// TwinCAT 3 PLC project External_Conveyor_system
// ProgramVersion: 3.1.4026.19
// libraries:
//   Tc2_EtherCAT, * (Beckhoff Automation GmbH)
//   Tc2_MC2, * (Beckhoff Automation GmbH)
//   Tc2_Standard, * (Beckhoff Automation GmbH)
//   Tc2_System, * (Beckhoff Automation GmbH)
//   Tc2_Utilities, * (Beckhoff Automation GmbH)
//   Tc3_Database, * (Beckhoff Automation GmbH)
//   Tc3_EventLogger, * (Beckhoff Automation GmbH)
//   Tc3_JsonXml, * (Beckhoff Automation GmbH)
//   Tc3_Module, * (Beckhoff Automation GmbH)
// project tree:
//   DUTs/EtherCAT模組/ MM540_Raw.TcDUT
//   DUTs/JOG用元素/ e_Site_Select.TcTLEO
//   DUTs/工單結構/ WorkOrder_Data.TcDUT
//   DUTs/變頻器IO/ VFD_E_IO.TcDUT
//   GVLs/ Axis.TcGVL, Config.TcGVL, Hmi_Web.TcGVL, Input.TcGVL, IO.TcGVL, Output.TcGVL, ProjectData.TcGVL, Safety.TcGVL
//   MSG/訊息列表/ MsgBuff.TcGVL
//   MSG/訊息格式/ MsgLevel.TcDUT, MsgStruct.TcDUT, MsgStruct_RAW.TcDUT
//   MSG/通知訊息/ MsgMain.TcPOU, MsgPush.TcPOU, uuidv7_g.TcPOU
//   / Note.TcPOU (excluded from build), PlcTask.TcTTO
//   POUs/ MAIN.TcPOU
//   POUs/功能塊/ ErrorCodeConver.TcPOU, pMsg.TcPOU, RW_Config.TcPOU
//   POUs/功能塊/EtherCat相關/ EtherCat_Driver_Reset.TcPOU, GetEtherSta.TcPOU
//   POUs/功能塊/字串處理功能塊/字串填充/ FILLSTRING.TcPOU
//   POUs/功能塊/字串處理功能塊/字串記憶/ WStrMem.TcPOU
//   POUs/功能塊/字串處理功能塊/字串連接/ StrConcat.TcPOU, WStrConcat.TcPOU
//   POUs/功能塊/資料庫 Postgre相關/動作資料/ ReadSQLData.TcPOU
//   POUs/功能塊/資料庫 Postgre相關/動作資料/相關結構/ e_db_steel_local.TcTLEO, e_db_steel_status.TcTLEO (not stored), sc_db_Set_Work_Order_WaitLoading_Pos.TcDUT, sc_db_Steel_Status.TcDUT
//   POUs/功能塊/資料庫 Postgre相關/記錄用/程式紀錄/ StepLog_Struct.TcDUT, Step_Log.TcPOU
//   POUs/動作流程控制/ Alignment_pos.TcDUT, FeedMain.TcPOU
//   POUs/動作流程控制/滾輪整料/ PullOver.TcPOU
//   POUs/安全控制/ MaBaseState.TcPOU
//   POUs/硬體控制/ AxisAction.TcPOU
//   POUs/硬體控制/出料滾輪/ ProductRoller.TcPOU
//   POUs/硬體控制/測高/ AxisBase.TcPOU, HeightMeasurer.TcPOU
//   POUs/硬體控制/油壓系統/ Hydraulic.TcPOU, Hydraulic_Action.TcDUT
//   POUs/硬體控制/測寬/ I_DisSensor.TcIO, OGD251_Decoder.TcPOU, Sensor.TcPOU
//   POUs/硬體控制/台車/ ActionMode.TcDUT, Axis_VFD.TcPOU, I_Axis.TcIO
//   POUs/硬體控制/台車/編碼器/ MM540.TcPOU
//   POUs/硬體控制/定位柱/ StopPin.TcPOU
//   POUs/硬體控制/進料滾輪/ FeedRoller.TcPOU
//   POUs/資料轉換/ HMI_WEB_dataConver.TcPOU
// (motion and I/O tree: see PLC project main)
// real-time tasks:
//   TASK Main_IO_Task: cycle T#2ms, priority 6, ADS port 353
//   TASK PlcTask: cycle T#10ms, priority 14, ADS port 350
//   TASK Conveyor: cycle T#10ms, priority 22, ADS port 355
// variable links:

CONFIGURATION External_Conveyor_system
    RESOURCE PLC ON TwinCAT3
        TASK PlcTask(INTERVAL := T#10ms, PRIORITY := 22);
        PROGRAM MAIN WITH PlcTask : MAIN;
    END_RESOURCE
END_CONFIGURATION

// ---- DUTs/EtherCAT模組/MM540_Raw.TcDUT
TYPE MM540_Raw :
STRUCT
	// 編碼器位置
	Inc AT %I*					: DINT;
	
	// 編碼器重設狀態
	Inc_Preload_Done AT %I*		: BOOL;
	
	// 編碼器 A相 錯誤
	Inc_Error_A AT %I*			: BOOL;
	
	// 編碼器 B相 錯誤
	Inc_Error_B AT %I*			: BOOL;
	
	// 編碼器 C相 錯誤
	Inc_Error_C AT %I*			: BOOL;
	
	// 編碼器1 AB相 錯誤
	Inc_Error_AB AT %I*			: BOOL;
	
	
	// 編碼器設定數值
	Inc_Preload_Value AT %Q*			: DINT;
	(*
	設定數值方式:
	0: Disabled
	1: Preload now
	2: Preload with next 0- impulse
	3: Preload with next DI0 rising edge
	4: Preload with next DI1 rising edge
	5: Preload with next DI2 rising edge
	6: Preload with next DI3 rising edge
	7: Preload with next DI0 falling edge
	8: Preload with next DI1 falling edge
	9: Preload with next DI2 falling edge
	10: Preload with next DI3 falling edge
	>10: Disabled
	*)
	// 編碼器1 設定數值方式
	Inc_Preload_Trigger AT %Q*				: USINT;
	
	// 1:數據無效 0:數據有效
	WcState AT %I*					: BOOL;
	
	// EtherCAT 狀態
	State AT %I*:UINT;
	
	// AMS位置
	addr 	AT %I*					: AMSADDR;
END_STRUCT
END_TYPE

// ---- DUTs/JOG用元素/e_Site_Select.TcTLEO
{attribute 'qualified_only'}
{attribute 'strict'}
{attribute 'to_string'}
TYPE e_Jog_Site_Select :
(
	Input_site := 0,
	Output_Site := 1
) INT ;
END_TYPE

// ---- DUTs/工單結構/WorkOrder_Data.TcDUT
// 專案資料結構
TYPE WorkOrder_Data :
STRUCT
	// 加工順序
	SN			: DINT;
	// 高
	Height		: LREAL;
	// 寬
	Width		: LREAL;
	// 素材編號 (uuid)
	steel_id	: STRING(36);
	//  在料架上等待的位置
	waitLoading_pos : LREAL;
END_STRUCT
END_TYPE

// ---- DUTs/變頻器IO/VFD_E_IO.TcDUT
TYPE VFD_E_IO :
STRUCT
	// 正轉 Output
	o_FWD : POINTER TO BOOL;
	
	// 逆轉 Output
	o_REV : POINTER TO BOOL;
	
	// 速度bit1 Output
	o_Speed1 : POINTER TO BOOL;
	
	// 速度bit2 Output
	o_Speed2 : POINTER TO BOOL;
	
	// 速度bit3 Output
	o_Speed3 : POINTER TO BOOL;
	
	// 重置 Output
	o_Reset : POINTER TO BOOL;
	
	// 運行中 Input
	i_Run : POINTER TO BOOL;
	
	// 發生錯誤 Input
	i_Error : POINTER TO BOOL;
END_STRUCT
END_TYPE

// ---- MSG/訊息格式/MsgLevel.TcDUT
{attribute 'qualified_only'}
{attribute 'strict'}
TYPE MsgLevel :
(
	Error	:= 4,
	Alarm	:= 2,
	Info	:= 1,
	None	:= 0
	
)INT;
END_TYPE

// ---- MSG/訊息格式/MsgStruct.TcDUT
{attribute 'pack_mode' := '1'} 
TYPE MsgStruct :
STRUCT
	// 訊息時間
	msgTIME		: DATE_AND_TIME;
	// 訊息等級
	Level		: MsgLevel;
	// 訊息號碼
	Number	: UINT;
	// 訊息附帶文字1
	MsgStr1	: WSTRING(80);
	// 訊息附帶文字2
	MsgStr2	: WSTRING(80);
	// 訊息全文
	raw_msg_str	: WSTRING(250);
END_STRUCT
END_TYPE

// ---- MSG/訊息格式/MsgStruct_RAW.TcDUT
{attribute 'pack_mode' := '1'} 
TYPE MsgStruct_RAW :
STRUCT
	// 訊息時間
	msgTIME		: DATE_AND_TIME;
	// 訊息等級
	Level		: MsgLevel;
	// 訊息號碼
	Number	: UINT;
	// 訊息附帶文字1
	MsgStr1	:  ARRAY[0..159] OF BYTE;
	// 訊息附帶文字2
	MsgStr2	: ARRAY[0..159] OF BYTE;
	// 訊息全文
	raw_msg_str	: ARRAY[0..499] OF BYTE;
END_STRUCT
END_TYPE

// ---- POUs/功能塊/資料庫 Postgre相關/動作資料/相關結構/e_db_steel_local.TcTLEO
{attribute 'qualified_only'}
{attribute 'strict'}
{attribute 'to_string'}
TYPE e_db_steel_local :
(
	holdingEntranceRack := 1, // 吊掛入料區
	entranceRack := 2, // 入料區
	machine := 10, // 機台內
	holdingExitRack := 20, // 吊掛出料區
	exitRack := 21 // 出料區
);
END_TYPE
//  exitRack = '21 '

// ---- POUs/功能塊/資料庫 Postgre相關/動作資料/相關結構/sc_db_Set_Work_Order_WaitLoading_Pos.TcDUT
TYPE sc_db_Set_Work_Order_WaitLoading_Pos :
STRUCT
	uuid : STRING(36);
	Pos : LREAL;
END_STRUCT
END_TYPE

// ---- POUs/功能塊/資料庫 Postgre相關/動作資料/相關結構/sc_db_Steel_Status.TcDUT
TYPE sc_db_Steel_Status :
STRUCT
	uuid : STRING(36);
	steel_status : STRING(80);
	steel_location : STRING(80);
END_STRUCT
END_TYPE

// ---- POUs/功能塊/資料庫 Postgre相關/記錄用/程式紀錄/StepLog_Struct.TcDUT
TYPE StepLog_Struct :
STRUCT
	step_number : DINT;
	created_at : LINT;
	program_name : STRING(80);
	extras_Srt : STRING(255) := '{}';
END_STRUCT
END_TYPE

// ---- POUs/動作流程控制/Alignment_pos.TcDUT
// 排列位置
TYPE Alignment_pos :
STRUCT
	// 分料開始位置 (搬運完成但未分料位置)
	Start : LREAL;
	// 分料結束位置 (推至分料位置)
	End : LREAL;
END_STRUCT
END_TYPE

// ---- POUs/硬體控制/油壓系統/Hydraulic_Action.TcDUT
{attribute 'qualified_only'}
{attribute 'strict'}
TYPE Hydraulic_Action :
(
	DoNothing	:= 0,
	Car_2_Up	:= 1,
	Car_2_Mid	:= 2,
	Car_2_Dn	:= 3,
	Pull_over	:= 4,
	UnPull		:= 5,
	Pull_over_Jog	:= 10
);
END_TYPE

// ---- POUs/硬體控制/台車/ActionMode.TcDUT
{attribute 'qualified_only'}
{attribute 'strict'}
TYPE ActionMode :
(
	DoNothing	:= 0,
	AbsMove		:= 1,
	RelMove		:= 2,
	Home		:= 3,
	Find		:= 4
);
END_TYPE

// ---- GVLs/Axis.TcGVL
VAR_GLOBAL
	
// 軸控制
// ============== 滾輪軸 ==============
	//  進料台車IO
	FeedCar_INV : VFD_E_IO;
	//  進料編碼器
	FeedCar_Enc : MM540;
	
	FeedCar : Axis_VFD;

// ============== 測高軸 ==============
	Axis_StepMoter: AXIS_REF;
	
	Axis_H_Measure: AxisBase;
	
	Override: LREAL := 100;
END_VAR

// ---- GVLs/Config.TcGVL
{attribute 'qualified_only'}
VAR_GLOBAL PERSISTENT
	// 靠邊感應器位置 
	SensorPos : ARRAY [0..15] OF UDINT := [2300,999999,6080,10230];

(* ===============台車===============*)
	// 台車間距
	Car_SetupPos : ARRAY [0..15] OF UDINT := [0,3700,7450,11200];
	
	// 臺車搬移平台寬度 1095mm
	FeedCar_Length : LREAL := 1095;
	
	// 臺車勾板寬度 25mm
	FeedCar_Pin_Length : LREAL := 25;
	
	// 台車橫移的編碼器比例
	FeedCar_Enc_Scal 			: LREAL := -0.025;
	
	// 臺車編碼器原點偏移 (編碼器值)
	FeedCar_Enc_Origin_offset 	: DINT := -880;
	
	// 臺車移動 高速 -> 中速 距離
	dis_to_MidSpeed : LREAL := 470;
	
	// 臺車移動 高速 -> 中速 距離
	dis_to_LowSpeed : LREAL := 80;
	
	// 臺車勾點-整料圓柱 位置  (測量寬度用)
	pos_CarPin_StopPoint		: LREAL := 1120;
	
	// 台車起點 (進料位置)
	pos_StartPoint				: LREAL := 60;
	
	// 台車 等待投料位置 (排列起點)
	pos_Workpiace_StanbyPoint	: LREAL := 1400;
	
	// 台車 投料位置 
	pos_Workpiace_FeedPoint	: LREAL := 2700;
	
	// 材料排列 間距
	dis_Alignment 				: LREAL := 100;
	
	// 材料容許誤差 倍率 (0-1 = 0 ~ 100%) 預設 10%
	Workpiace_Err_size 				: LREAL := 0.1;
	
(* =============== 測高 =============== *)
	// 高基準面位置
	H_Measure_ZeroPoint : LREAL := 642.62;
	
(* =============== 測寬感應器 =============== *)
	// 寬基準面位置
	W_Measure_ZeroPoint : LREAL := 1253;
	
	

END_VAR

// ---- GVLs/Hmi_Web.TcGVL
{attribute 'qualified_only'}
VAR_GLOBAL
(*==================== Jog模式====================*)
	// 料架選擇
	Site_Select : e_Jog_Site_Select;
	
	// 料架速度 (0:高速 1:低速)
	Speed_Select : INT;
	
	// 指定橫移料架
	Module_Select : INT;
	
	// 動力滾輪正轉反饋
	Roller_Fwd_S : BOOL;
	// 動力滾輪反轉反饋
	Roller_Rev_S : BOOL;
	
	// 動力滾輪正轉
	Roller_Fwd : BOOL;
	// 動力滾輪反轉
	Roller_Rev : BOOL;
	
	
	// 動力滾輪上升
	Roller_Up_S : BOOL;
	// 動力滾輪下降
	Roller_Down_S : BOOL;
	
	// 動力滾輪上升
	Roller_Up : BOOL;
	// 動力滾輪下降
	Roller_Down : BOOL;
	
	// 橫移台車位置
	Car_Pos : LREAL;
	// 橫移台車正轉
	Car_Fwd_S : BOOL;
	// 橫移台車反轉
	Car_Rev_S : BOOL;
	
	// 橫移台車正轉
	Car_Fwd : BOOL;
	// 橫移台車反轉
	Car_Rev : BOOL;
	
	
	// 橫移台車上升
	Car_Up_S : BOOL;
	// 橫移台車下降
	Car_Down_S : BOOL;
	
	// 橫移台車上升
	Car_Up : BOOL;
	// 橫移台車下降
	Car_Down : BOOL;
	
	
	// 定位柱上升
	StopPin_Up_S : BOOL;
	// 定位柱下降
	StopPin_Down_S : BOOL;
	
	// 定位柱上升
	StopPin_Up : BOOL;
	// 定位柱下降
	StopPin_Down : BOOL;


	// 橫移台車上升
	Pull_over_Push_S : BOOL;

	// 靠邊推
	Pull_over_Push : BOOL;
END_VAR

// ---- GVLs/Input.TcGVL
VAR_GLOBAL
	// 暫停
	Pause					AT %I*	: BOOL;
	
	// 進料機 啟動
	Feed_Start				AT %I*	: BOOL;
	
	// 進料機 執行動作
	Feed_Mode				AT %I*	: INT;
	
	// 進料機 進料的專案UUID
	Feed_WorkOrder_UUID		AT %I*	: STRING(36);
	
	// 進料機 啟動
	Feed_Enable				AT %I*	: BOOL;
	
	// 進料機 重置
	Feed_Reset				AT %I*	: BOOL;
	
	// 靠邊 模式執行
	PullOver_Start			AT %I*	: BOOL;
	
	// 進料滾輪啟動
	In_Moter_Start 			AT %I*	: BOOL;
	
	// 出料滾輪啟動
	Out_Moter_Start 		AT %I*	: BOOL;
END_VAR

// ---- GVLs/IO.TcGVL
{attribute 'qualified_only'}
VAR_GLOBAL
{region "============= EL1409_1 ============="}
	//
	i101 AT %I*: BOOL;
	// 入料側油壓馬達過載檢知
	i102 AT %I*: BOOL;
	// 抽油循環馬達
	i103 AT %I*: BOOL;
	// 入料側油壓馬達過載檢知
	i104 AT %I*: BOOL;
	// 入料側橫移馬達過載1檢知
	i105 AT %I*: BOOL;
	// 入料側橫移馬達過載2檢知
	i106 AT %I*: BOOL;
	// 入料側橫移變頻器運轉
	i107 AT %I*: BOOL;
	// 入料側橫移變頻器無異常
	i108 AT %I*: BOOL;
	// 入料側上浮滾輪馬達過載1檢知
	i109 AT %I*: BOOL;
	// 入料側上浮滾輪馬達過載2檢知
	i110 AT %I*: BOOL;
	// 入料側上浮滾輪馬達過載3檢知
	i111 AT %I*: BOOL;
	// 入料側上浮滾輪馬達過載4檢知
	i112 AT %I*: BOOL;
	// 出口上浮滾輪停止
	i113 AT %I*: BOOL;
	// 出口有無料檢測1
	i114 AT %I*: BOOL;
	// 出口有無料檢測2
	i115 AT %I*: BOOL;
	// 
	i116 AT %I*: BOOL;
 {endregion}
{region "============= EL1409_2 ============="}
	// 入料側橫移台車升降1上限
	i201 AT %I*: BOOL;
	// 入料側橫移台車升降1中限
	i202 AT %I*: BOOL;
	// 入料側橫移台車升降1下限
	i203 AT %I*: BOOL;
	// 入料側橫移台車升降2上限
	i204 AT %I*: BOOL;
	// 入料側橫移台車升降2中限
	i205 AT %I*: BOOL;
	// 入料側橫移台車升降2下限
	i206 AT %I*: BOOL;
	// 入料側橫移台車升降3上限
	i207 AT %I*: BOOL;
	// 入料側橫移台車升降3中限
	i208 AT %I*: BOOL;
	// 入料側橫移台車升降3下限
	i209 AT %I*: BOOL;
	// 入料側橫移台車升降4上限
	i210 AT %I*: BOOL;
	// 入料側橫移台車升降4中限
	i211 AT %I*: BOOL;
	// 入料側橫移台車升降4下限
	i212 AT %I*: BOOL;
	// 入料側橫移台車原點
	i213 AT %I*: BOOL;
	// 
	i214 AT %I*: BOOL;
	// 
	i215 AT %I*: BOOL;
	// 
	i216 AT %I*: BOOL;
{endregion}
{region "============= EL1409_3 ============="}
	// 入料側整料圓柱1下限
	i301 AT %I*: BOOL;
	// 入料側整料圓柱1上限
	i302 AT %I*: BOOL;
	// 入料側整料圓柱1材料定位
	i303 AT %I*: BOOL;
	// 入料側整料圓柱2下限
	i304 AT %I*: BOOL;
	// 入料側整料圓柱2上限
	i305 AT %I*: BOOL;
	// 入料側整料圓柱2材料定位
	i306 AT %I*: BOOL;
	// 入料側整料圓柱3下限
	i307 AT %I*: BOOL;
	// 入料側整料圓柱3上限
	i308 AT %I*: BOOL;
	// 入料側整料圓柱3材料定位
	i309 AT %I*: BOOL;
	// 入料側整料圓柱4下限
	i310 AT %I*: BOOL;
	// 入料側整料圓柱4上限
	i311 AT %I*: BOOL;
	// 入料側整料圓柱4材料定位
	i312 AT %I*: BOOL;
	// 出口滾輪
	i313 AT %I*: BOOL;
	// 測高上限原點
	i314 AT %I*: BOOL;
	// 出料側上浮滾輪升降 上限(滾輪下)
	i315 AT %I*: BOOL;
	// 出料側上浮滾輪升降 下限(滾輪上)
	i316 AT %I*: BOOL;
 {endregion}
{region "============= EL1409_4 ============="}
	// 入料側靠邊1原點
	i401 AT %I*: BOOL;
	// 入料側靠邊1材料定位檢知
	i402 AT %I*: BOOL;
	// 入料側靠邊2原點
	i403 AT %I*: BOOL;
	// 入料側靠邊2材料定位檢知
	i404 AT %I*: BOOL;
	// 入料側靠邊3原點
	i405 AT %I*: BOOL;
	// 入料側靠邊3材料定位檢知
	i406 AT %I*: BOOL;
	// 入料側靠邊4原點
	i407 AT %I*: BOOL;
	// 入料側靠邊4材料定位檢知
	i408 AT %I*: BOOL;
	// 入料側滾輪1 離合器 分離
	i409 AT %I*: BOOL;
	// 入料側滾輪1 離合器 結合
	i410 AT %I*: BOOL;
	// 入料側上浮滾輪升降2 下限(滾輪上)
	i411 AT %I*: BOOL;
	// 入料側上浮滾輪升降2 上限(滾輪下)
	i412 AT %I*: BOOL;
	// 
	i413 AT %I*: BOOL;
	// 
	i414 AT %I*: BOOL;
	// 
	i415 AT %I*: BOOL;
	// 
	i416 AT %I*: BOOL;
 {endregion}
	  
	 
{region "============= EL2409_7 ============="}
	// 入料側油壓馬達啟動
	q101 AT %Q*: BOOL;
	// 入料側上浮滾輪(全) 反轉
	q102 AT %Q*: BOOL;
	// 入料側上浮滾輪(全) 正轉
	q103 AT %Q*: BOOL;
	// 入料側橫移台車變頻器正轉 (往靠邊)
	q104 AT %Q*: BOOL;
	// 入料側橫移台車變頻器反轉 (往原點)
	q105 AT %Q*: BOOL;
	// 入料側橫移台車變頻器多段速01
	q106 AT %Q*: BOOL;
	// 入料側橫移台車變頻器多段速02
	q107 AT %Q*: BOOL;
	// 入料側橫移台車變頻器多段速03(未設定)
	q108 AT %Q*: BOOL;
	// 
	q109 AT %Q*: BOOL;
	// 
	q110 AT %Q*: BOOL;
	// 
	q111 AT %Q*: BOOL;
	// 
	q112 AT %Q*: BOOL;
	// 
	q113 AT %Q*: BOOL;
	// 出口側上浮滾輪反轉
	q114 AT %Q*: BOOL;
	// 出口側上浮滾輪正轉
	q115 AT %Q*: BOOL;
	// 
	q116 AT %Q*: BOOL;
{endregion}
{region "============= EL2409_8 ============="}
	// 入料側橫移台車1上升
	q201 AT %Q*: BOOL;
	// 入料側橫移台車1下降
	q202 AT %Q*: BOOL;
	// 入料側橫移台車2上升
	q203 AT %Q*: BOOL;
	// 入料側橫移台車2下降
	q204 AT %Q*: BOOL;
	// 入料側橫移台車3上升
	q205 AT %Q*: BOOL;
	// 入料側橫移台車3下降
	q206 AT %Q*: BOOL;
	// 入料側橫移台車4上升
	q207 AT %Q*: BOOL;
	// 入料側橫移台車4下降
	q208 AT %Q*: BOOL;
	// 入料側整料圓柱1上升
	q209 AT %Q*: BOOL;
	// 入料側整料圓柱1下降
	q210 AT %Q*: BOOL;
	// 入料側整料圓柱2上升
	q211 AT %Q*: BOOL;
	// 入料側整料圓柱2下降
	q212 AT %Q*: BOOL;
	// 入料側整料圓柱3上升
	q213 AT %Q*: BOOL;
	// 入料側整料圓柱3下降
	q214 AT %Q*: BOOL;
	// 入料側整料圓柱4上升
	q215 AT %Q*: BOOL;
	// 入料側整料圓柱4下降
	q216 AT %Q*: BOOL;
{endregion}
{region "============= EL2409_9 ============="}
	// 入料側油壓總閥
	q301 AT %Q*: BOOL;
	// 入料側油壓靠邊閥
	q302 AT %Q*: BOOL;
	// 入料側測高上升
	q303 AT %Q*: BOOL;
	// 入料側測高下降
	q304 AT %Q*: BOOL;
	// 出口側出料滾輪1下降
	q305 AT %Q*: BOOL;
	// 出口側出料滾輪1上升
	q306 AT %Q*: BOOL;
	// 入料側變頻器異常清除
	q307 AT %Q*: BOOL;
	// 
	q308 AT %Q*: BOOL;
	// 入料側進料滾輪1 離合器接合
	q309 AT %Q*: BOOL;
	// 入料側進料滾輪1 離合器分離
	q310 AT %Q*: BOOL;
	// 入料側進料滾輪2 上升
	q311 AT %Q*: BOOL;
	// 入料側進料滾輪2 下降
	q312 AT %Q*: BOOL;
	// 
	q313 AT %Q*: BOOL;
	// 
	q314 AT %Q*: BOOL;
	// 
	q315 AT %Q*: BOOL;
	// 
	q316 AT %Q*: BOOL;
{endregion}
END_VAR

// ---- GVLs/Output.TcGVL
VAR_GLOBAL
	// 進料機 動作中
	Feed_bBuzy						AT %Q*	: BOOL;
	// 進料機 動作完成
	Feed_bDone 						AT %Q*	: BOOL;
	// 進料機 發生錯誤
	Feed_bError 					AT %Q*	: BOOL;
	
	// 進料材料寬度
	Feed_Workpiace_W 				AT %Q*	: LREAL;
	
	// 進料材料高度
	Feed_Workpiace_H 				AT %Q*	: LREAL;
	
	// 執行中的動作
	ActionMode_Now 					AT %Q*	: UINT;
	
	
	// 靠邊 動作中
	PullOver_bBuzy					AT %Q*	: BOOL;
	// 靠邊  動作完成
	PullOver_bDone 					AT %Q*	: BOOL;
	// 靠邊  發生錯誤
	PullOver_bError 				AT %Q*	: BOOL;
	
	
	// 靠邊光電感應器
	in_Pos_sensor					AT %Q*	: WORD;
	
	// 靠邊光電感應器
	Out_Pos_sensor					AT %Q*	: WORD;
	
	// 進料滾輪啟動
	In_Moter_Running 				AT %Q*	: BOOL;
	// 進料滾輪錯誤
	In_Moter_Error 					AT %Q*	: BOOL;
	
	
	// 出料滾輪啟動
	Out_Moter_Running 				AT %Q*	: BOOL;
	// 出料滾輪錯誤
	Out_Moter_Error 				AT %Q*	: BOOL;
	
	
END_VAR

// ---- GVLs/ProjectData.TcGVL
{attribute 'qualified_only'}
VAR_GLOBAL
	// 人工置料完成(已註冊)數量
	WorkOrder_Nunber_At_holding : UINT;
	
	WorkOrder_At_holding 	: ARRAY [0..9] OF WorkOrder_Data;
	
	WorkOrder_Nunber_At_waitLoading : UINT;
	
	WorkOrder_At_waitLoading 	: ARRAY [0..9] OF WorkOrder_Data;
	
	WorkOrder_Nunber_At_Machining : UINT;
END_VAR

// ---- GVLs/Safety.TcGVL

VAR_GLOBAL
	// 緊急停止
	Estop: BOOL;	
	// 光柵
	Door: BOOL;
	
	SystemError :BOOL;
	
	SystemAlarm :BOOL;
	
	
	close_Air_Pressure_Check:bool;
	
	//關閉前方光柵
	close_Door_Bad:BOOL;
	//關閉臺車出入口光柵
	close_Door_Car_Gate:BOOL;
	//關閉臺車周圍光柵
	close_Door_Car_Around:BOOL;
	
	//關閉鏈條斷裂檢
	close_Chain_Break_Check: BOOL;
	
	// 真空壓力感應器
	VacuumSensor: BOOL;
END_VAR

// ---- MSG/訊息列表/MsgBuff.TcGVL
{attribute 'qualified_only'}
VAR_GLOBAL
	// 儲列使用計數器
	evenNumber		: UDINT;
	
	DoneNumber 		: UDINT;

	messageList : ARRAY[0..15] OF MsgStruct;
	
// SQL 執行命令型
_fb_PLCDBCmdEvt : FB_PLCDBCmdEvt(sNetID:= '', tTimeout:= T#5S );

	systime         : FB_LocalSystemTime;
	currentTime     : DT;
END_VAR

// ---- POUs/硬體控制/測寬/I_DisSensor.TcIO
INTERFACE I_DisSensor

PROPERTY Distance : REAL
GET
END_GET
END_PROPERTY

END_INTERFACE

// ---- POUs/硬體控制/台車/I_Axis.TcIO
INTERFACE I_Axis

METHOD AbsMove : BOOL
VAR_INPUT
	// 目標位置
	_Position : LREAL;
	// 移動速度
	_Velocity : LREAL := 0;
END_VAR
END_METHOD

PROPERTY Buzy : bool
GET
END_GET
END_PROPERTY

PROPERTY Done : bool
GET
END_GET
END_PROPERTY

PROPERTY Error : bool
GET
END_GET
END_PROPERTY

METHOD Homing : BOOL
VAR_INPUT
END_VAR
END_METHOD

METHOD PowerOff : BOOL
VAR_INPUT
END_VAR
END_METHOD

METHOD PowerOn : BOOL
VAR_INPUT
END_VAR
END_METHOD

METHOD RelMove : BOOL
VAR_INPUT
	// 目標距離
	_Position : LREAL;
	
	// 移動速度
	_Velocity : LREAL := 0;
END_VAR
END_METHOD

METHOD SetLimit : BOOL
VAR_INPUT
END_VAR
END_METHOD

METHOD Stop : BOOL
VAR_INPUT
END_VAR
END_METHOD

END_INTERFACE

// ---- POUs/MAIN.TcPOU
PROGRAM MAIN
VAR
	
	i : INT;

	val: ARRAY [0..100] OF REAL;
	
	postmp: REAL;
END_VAR

MaBaseState();

// 測距感應器
Sensor();

// 測高機構
HeightMeasurer();

// 定位圓柱
StopPin();

AxisAction();

FeedMain();

// 進料滾輪
FeedRoller();
// 出料滾輪
ProductRoller();

Hydraulic();

ReadSQLData();

PullOver();

HMI_WEB_dataConver();

MsgMain();

END_PROGRAM

// ---- POUs/安全控制/MaBaseState.TcPOU
PROGRAM MaBaseState
VAR
	trig1: R_TRIG;
	trig2: F_TRIG;
	tmr01 : TON;
END_VAR

E_Stop();

trig1(CLK:= Input.Feed_Reset);
trig2(CLK:= Input.Feed_Reset);

tmr01(IN:=SystemError, PT := T#2S);

IF trig1.Q THEN
	SystemError := TRUE;
END_IF

IF trig2.Q THEN
	SystemError := FALSE;
END_IF

ACTION E_Stop:
//	========================================
//					緊急停止				
//	========================================

// Estop := NOT(IO.i101);
// 
// //// 緊急停止
// E_stop_trig1(clk:=IO.i616); 
// IF E_stop_trig1.Q THEN
// 	pMsg.Push_Error("緊急停止");
// END_IF

//E_stop_trig2(clk:=io3.X001); 
//IF E_stop_trig2.Q THEN
//	pMsg.Push_Error("緊急停止 倉儲面板");
//END_IF

//E_stop_trig2(clk:=io0.X002 AND io0.X003); 
//IF E_stop_trig2.Q THEN
//	pMsg.Push_Error("緊急停止 台車面板");
//END_IF

//E_stop_trig3(clk:=io0.X101); 
//IF E_stop_trig3.Q THEN
//	pMsg.Push_Error("緊急停止 台車");
//END_IF
END_ACTION

END_PROGRAM

// ---- POUs/硬體控制/測寬/Sensor.TcPOU
PROGRAM Sensor
VAR
	sensor	: OGD251_Decoder := (DisableSeosor := false);
	
	tmp_value: LREAL;
END_VAR

VAR_OUTPUT
	MeasureValue : LREAL;
END_VAR

// 測距感應器
sensor();

tmp_value := config.W_Measure_ZeroPoint - sensor.fDistance;

IF sensor.fDistance <> 0 THEN
	MeasureValue := tmp_value;
ELSE
	MeasureValue := 0;
END_IF

METHOD Measure : BOOL
VAR_INPUT
END_VAR
MeasureValue := config.W_Measure_ZeroPoint - sensor.fDistance;
END_METHOD

END_PROGRAM

// ---- POUs/硬體控制/測寬/OGD251_Decoder.TcPOU
FUNCTION_BLOCK OGD251_Decoder IMPLEMENTS I_DisSensor
VAR_INPUT
	// 關閉感應器
	DisableSeosor :	BOOL;
END_VAR
VAR_OUTPUT
	// 距離 (單位:mm)
	fDistance : REAL;
	// 裝置狀態正常
	SSC1_1			:BOOL;
	// 裝置狀態正常
	bDevice_is_OK			:BOOL;
	// 需要維護
	bMaintenance_required	:BOOL;
	// 超出測量距離
	bOut_of_specification	:BOOL;
	// 檢查功能
	bFunctional_check		:BOOL;
	// 錯誤
	bFailure				:BOOL;
	// 距離比例(單位:公尺)
	iScale_Distance			:INT;
END_VAR
VAR
	// 原始資料輸入
	in_RawData AT %I* : ARRAY [0..7] OF USINT;
	// 原始資料輸出
	out_rawdata AT %Q* :USINT;	
	
	

	DistanceTmp : WORD;
	tmpStatus : WORD;
	tmpStatus2 : WORD;
	tmpStatus3 : POINTER TO SINT;
	tmpfDistance : SINT;
END_VAR

DistanceTmp := USINT_TO_WORD(in_RawData[0]);

DistanceTmp := ROL(DistanceTmp, 8) + USINT_TO_WORD(in_RawData[1]);


// 數值比例 (單位:公尺)
tmpStatus3 := ADR(in_RawData[2]);




IF (DistanceTmp = 16#7FF8) OR (DistanceTmp = 16#8008) OR (DistanceTmp = 16#7FFC) THEN
	fDistance := 0;
ELSE
	// 距離 = 感應器RAW值 X 10^單位值 X 1000(將 m 轉為 mm)
	fDistance := LREAL_TO_REAL(DistanceTmp * EXPT(10, tmpStatus3^) * 1000);
END_IF

tmpStatus := ROR(in_RawData[3] AND 16#F0, 4);

SSC1_1 := (in_RawData[3] AND 16#1) = 1;

bDevice_is_OK := tmpStatus = 0;
bMaintenance_required := tmpStatus = 1;
bOut_of_specification := tmpStatus = 2;
bFunctional_check := tmpStatus = 3;
bFailure := tmpStatus = 4;

tmpStatus2 := 0;
tmpStatus2.0 := DisableSeosor;

out_rawdata := WORD_TO_USINT(tmpStatus2);

PROPERTY Distance : REAL
GET
Distance := fDistance;
END_GET
END_PROPERTY

END_FUNCTION_BLOCK

// ---- POUs/硬體控制/測高/HeightMeasurer.TcPOU
PROGRAM HeightMeasurer
VAR
	// 程式流程
	step : INT;
	
	// 已歸零
	bHome: BOOL;
	
	tmr01 : TON;
	// 位置
	_pos: LREAL;
	// 上次的位置 計算速度用
	_lastPos: LREAL;
	// 速度
	_speed: LREAL;
	bBoot: BOOL := true;
	tmpTargetPos: LREAL;
	
	tmp_MeasurePos: LREAL;
END_VAR

VAR_OUTPUT
	bDone : BOOL;
	bBuzy : BOOL;
	bError : BOOL;
	MeasureValue : Lreal;
END_VAR

IF bBoot THEN
	initAction();
	bBoot := FALSE;
END_IF

Axis.Axis_H_Measure(outLimiter := TRUE, inLimiter := NOT IO.i314, origin := IO.i314);

Step_000_Measure();
Step_100_Measure_Error();
Step_3_homming();

bBuzy := step > 0 AND step < 10000;
bError := step > 10000;

IF bError OR bBuzy THEN
	bDone := FALSE;
END_IF

output.Feed_Workpiace_W := MeasureValue;

Axis.Axis_H_Measure();

tmrAct();

PROPERTY at_Home : bool
GET
at_Home := IO.i314;
END_GET
END_PROPERTY

METHOD Homing : BOOL
VAR_INPUT
END_VAR
step := 300;
END_METHOD

METHOD initAction : BOOL
VAR_INPUT
END_VAR
Axis.Axis_H_Measure.Name := "H_Measure";

Axis.Axis_H_Measure.Axis1 REF= Axis.Axis_StepMoter;
END_METHOD

METHOD Measure : BOOL
VAR_INPUT
END_VAR
step := 1;
END_METHOD

ACTION Step_000_Measure:
CASE step OF
	1:
		
		step := step + 1;
		
	2:
		IF NOT Axis.Axis_H_Measure.bHome THEN
			step := 10;
		ELSE
			step := 30;
		END_IF
		
	10:
		Axis.Axis_H_Measure.Homing();
		step := step + 1;
	
	11:
		IF  Axis.Axis_H_Measure.bBuzy OR Axis.Axis_H_Measure.bError THEN
			step := step + 1;
		END_IF
		
	12:
		IF Axis.Axis_H_Measure.bDone THEN
			step := step + 1;
		ELSIF Axis.Axis_H_Measure.bError THEN
			step := step + 10000;
		END_IF
		
	13:
		step := 30;
		
	20:
		IF ProjectData.WorkOrder_At_holding[0].Height > 0 THEN
			tmpTargetPos := config.H_Measure_ZeroPoint - (ProjectData.WorkOrder_At_holding[0].Height + 50);
			step := step + 1;
		ELSE
			step := 30;
		END_IF
		
	21:
		IF tmpTargetPos > 0 THEN
			Axis.Axis_H_Measure.AbsMove(tmpTargetPos, 200);
			step := step + 1;
		ELSE
			step := 30;
		END_IF
		
	22:
		IF  Axis.Axis_H_Measure.bBuzy OR Axis.Axis_H_Measure.bError THEN
			step := step + 1;
		END_IF
		
	23:
		IF Axis.Axis_H_Measure.bDone THEN
			tmr01.IN := FALSE;
			step := step + 1;
		ELSIF Axis.Axis_H_Measure.bError THEN
			tmr01.IN := FALSE;
			step := step + 10000;
		END_IF
		
	24:
		step := 30;
		
	30:
		Axis.Axis_H_Measure.AbsMove(config.H_Measure_ZeroPoint, 100);
		step := step + 1;
		
	31:
		IF  Axis.Axis_H_Measure.bBuzy OR Axis.Axis_H_Measure.bError THEN
			step := step + 1;
		END_IF
		
	32:
		tmr01.PT := T#500MS;
		tmr01.IN := abs(Axis.Axis_H_Measure.Axis1.NcToPlc.ActVelo) < 1;
		
		IF tmr01.Q THEN
			Axis.Axis_H_Measure.Stop();
			tmr01.IN := FALSE;
			step := step + 1;
		ELSIF Axis.Axis_H_Measure.bDone THEN
			tmr01.IN := FALSE;
			step := 100;
		ELSIF Axis.Axis_H_Measure.bError THEN
			tmr01.IN := FALSE;
			step := step + 10000;
		END_IF
		
	33:
		IF NOT Axis.Axis_H_Measure.bBuzy THEN
			step := step + 1;
		END_IF
		
	34:
		step := 40;
		
	40:
		MeasureValue := config.H_Measure_ZeroPoint - Axis.Axis_H_Measure.fPos;
		tmp_MeasurePos := Axis.Axis_H_Measure.fPos;
		step := step + 1;
		
	41:
		Axis.Axis_H_Measure.AbsMove(-5, 200);
		step := step + 1;
		
	42:
		IF  Axis.Axis_H_Measure.bBuzy OR Axis.Axis_H_Measure.bError THEN
			step := step + 1;
		END_IF
		
	43:
		IF Axis.Axis_H_Measure.bDone OR (tmp_MeasurePos - Axis.Axis_H_Measure.fPos) > 50  THEN
			step := step + 1;
		ELSIF Axis.Axis_H_Measure.bError THEN
			step := step + 10000;
		END_IF
		
	44:
		step := 90;
	
	90:
		bdone := TRUE;
		step := 0;
END_CASE
END_ACTION

ACTION Step_100_Measure_Error:
CASE step OF
	100:
		step := 110;
		
	
	110:
		Axis.Axis_H_Measure.AbsMove(-5, 200);
		step := step + 1;
		
	111:
		IF  Axis.Axis_H_Measure.bBuzy OR Axis.Axis_H_Measure.bError THEN
			step := step + 1;
		END_IF
		
	112:
		IF Axis.Axis_H_Measure.bDone THEN
			step := step + 1;
		ELSIF Axis.Axis_H_Measure.bError THEN
			step := step + 10000;
		END_IF
		
	113:
		step := 190;
	
	190:
		pMsg.Push_Error("未檢測到工件");
		step := step + 10000;
END_CASE
END_ACTION

ACTION Step_3_homming:
CASE step OF
	300:
		IF Axis.Axis_H_Measure.bHome THEN
			step := 380;
		ELSE
			step := 310;
		END_IF
		
	310:
		Axis.Axis_H_Measure.Homing();
		step := step + 1;
	
	311:
		IF  Axis.Axis_H_Measure.bBuzy OR Axis.Axis_H_Measure.bError THEN
			step := step + 1;
		END_IF
		
	312:
		IF Axis.Axis_H_Measure.bDone THEN
			step := step + 1;
		ELSIF Axis.Axis_H_Measure.bError THEN
			step := step + 10000;
		END_IF
		
	313:
		step := 380;

	380:
		Axis.Axis_H_Measure.AbsMove(-5, 100);
		step := step + 1;
		
	381:
		IF  Axis.Axis_H_Measure.bBuzy OR Axis.Axis_H_Measure.bError THEN
			step := step + 1;
		END_IF
		
	382:
		IF Axis.Axis_H_Measure.bDone THEN
			step := step + 1;
		ELSIF Axis.Axis_H_Measure.bError THEN
			step := step + 10000;
		END_IF
		
	383:
		step := 390;
		
	390:
		bhome := TRUE;
		bdone := TRUE;
		step := 0;
		
END_CASE
END_ACTION

ACTION tmrAct:
tmr01();
END_ACTION

END_PROGRAM

// ---- POUs/功能塊/pMsg.TcPOU
PROGRAM pMsg
VAR
	msg: MsgPush;
END_VAR

METHOD PUBLIC Push_Alarm : BOOL
VAR_INPUT
	STR : WSTRING;
END_VAR
msg.iMessageId := 0;
msg.msgeLevel := MsgLevel.Alarm;
msg.sMessageStr1:=STR;
msg();
END_METHOD

METHOD PUBLIC Push_Alarm_NoPause : BOOL
VAR_INPUT
	STR : WSTRING;
END_VAR
msg.iMessageId := 0;
msg.msgeLevel := MsgLevel.Alarm;
msg.sMessageStr1:=STR;
msg();
END_METHOD

METHOD PUBLIC Push_Error : BOOL
VAR_INPUT
	STR : WSTRING;
END_VAR
msg.iMessageId := 0;
msg.msgeLevel := MsgLevel.Error;
msg.sMessageStr1:=STR;
SystemError := TRUE;
msg();
END_METHOD

METHOD PUBLIC Push_Info : BOOL
VAR_INPUT
	STR : WSTRING;
	
END_VAR
msg.iMessageId := 0;
msg.msgeLevel := MsgLevel.Info;
msg.sMessageStr1:=STR;
msg();
END_METHOD

END_PROGRAM

// ---- MSG/通知訊息/MsgPush.TcPOU
FUNCTION_BLOCK MsgPush
VAR_INPUT
	// 事件等級(MessageLevel.info:訊息、.Alarm:警告、.Error:錯誤)
	msgeLevel: MsgLevel;
	// 訊息編號
	iMessageId: UINT;
	// 訊息插入文字1
	sMessageStr1: WSTRING(80) := "";
	// 訊息插入文字2
	sMessageStr2: WSTRING(80) := "";
	
END_VAR

VAR
	msg		: MsgStruct;
	
	MsgNum			: USINT;
	
	
	
	
	
END_VAR
VAR_OUTPUT
	bDone: BOOL;
	nState : INT;
END_VAR

MsgNum := ULINT_TO_USINT(MsgBuff.evenNumber MOD 16);



//MsgBuff.messageList[MsgNum].MsgTime := 	FILETIME_TO_DT(currentTime);
//MsgBuff.messageList[MsgNum].Level :=	msgeLevel;
//MsgBuff.messageList[MsgNum].Number :=	iMessageId;
//MsgBuff.messageList[MsgNum].MsgStr1 :=	sMessageStr1;
//MsgBuff.messageList[MsgNum].MsgStr2 :=	sMessageStr2;
//MsgBuff.messageList[MsgNum].Sn :=		MsgBuff.evenNumber;
MsgBuff.evenNumber := MsgBuff.evenNumber + 1;

bDone := FALSE;

msg.MsgTime := 	MsgBuff.currentTime;
msg.Level :=	msgeLevel;
msg.Number :=	iMessageId;
msg.MsgStr1 :=	sMessageStr1;
msg.MsgStr2 :=	sMessageStr2;
msg.raw_msg_str := sMessageStr1;

MsgBuff.messageList[MsgNum] := msg;

END_FUNCTION_BLOCK

// ---- POUs/硬體控制/定位柱/StopPin.TcPOU
PROGRAM StopPin
VAR
	// 程式流程
	step : INT;
	
	Module_Select : WORD;
	
	tmr01 : TON;
END_VAR

VAR_OUTPUT
	bDone : BOOL;
	bBuzy : BOOL;
	bError : BOOL;
END_VAR


Step_1_Up();

Step_2_Down();

bBuzy := step > 0 AND step < 10000;
bError := step > 10000;

IF bError OR bBuzy THEN
	bDone := FALSE;
END_IF

tmrAct();

METHOD Down : BOOL
VAR_INPUT
	// 動作的台車 bit0:台車1、bit0:台車2、bit0:台車3、bit0:台車4
	Action_Select : WORD := 0;
END_VAR
IF Action_Select = 0 THEN
	Module_Select := 255;
ELSE
	Module_Select := Action_Select;
END_IF
step := 200;
END_METHOD

ACTION Step_1_Up:
CASE step OF
	100: // 圓柱上升
		io.q209 := Module_Select.0;
		io.q210 := FALSE;
		io.q211 := Module_Select.1;
		io.q212 := FALSE;
		io.q213 := Module_Select.2;
		io.q214 := FALSE;
		io.q215 := Module_Select.3;
		io.q216 := FALSE;
		
		tmr01.in := TRUE;
		tmr01.PT := T#15S;
		
		step := step + 1;
		
	101: // 確定要上升的圓柱都已到定位圓柱上升
		IF tmr01.q OR
		 	(
				(NOT Module_Select.0 OR io.i302) AND 
				(NOT Module_Select.1 OR io.i305) AND 
				(NOT Module_Select.2 OR io.i308) AND 
				(NOT Module_Select.3 OR io.i311)
			)
		THEN
			io.q209 := FALSE;
			io.q211 := FALSE;
			io.q213 := FALSE;
			io.q215 := FALSE;
			
			tmr01.in := FALSE;
			
			IF (NOT Module_Select.0 OR io.i302) AND 
				(NOT Module_Select.1 OR io.i305) AND 
				(NOT Module_Select.2 OR io.i308) AND 
				(NOT Module_Select.3 OR io.i311)
			THEN
				step := step + 1;
			ELSIF tmr01.q THEN
				step := step + 10000;
			END_IF
			
		END_IF	
		
	102:
		bdone := TRUE;
		step := 0;
	
		
		
END_CASE
END_ACTION

ACTION Step_2_Down:
CASE step OF
	200: // 圓柱下降
		io.q209 := FALSE;
		io.q210 := Module_Select.0;
		io.q211 := FALSE;
		io.q212 := Module_Select.1;
		io.q213 := FALSE;
		io.q214 := Module_Select.2;
		io.q215 := FALSE;
		io.q216 := Module_Select.3;
		
		tmr01.in := TRUE;
		tmr01.PT := T#15S;
		
		step := step + 1;
		
	201: // 確定所有圓柱 已下降
		IF tmr01.q OR 
			(
				(NOT Module_Select.0 OR io.i301) AND 
				(NOT Module_Select.1 OR io.i304) AND 
				(NOT Module_Select.2 OR io.i307) AND 
				(NOT Module_Select.3 OR io.i310)
			)
		 THEN
			io.q210 := FALSE;
			io.q212 := FALSE;
			io.q214 := FALSE;
			io.q216 := FALSE;
			
			tmr01.in := FALSE;
			
			IF (NOT Module_Select.0 OR io.i301) AND 
				(NOT Module_Select.1 OR io.i304) AND 
				(NOT Module_Select.2 OR io.i307) AND 
				(NOT Module_Select.3 OR io.i310)
			THEN
				step := step + 1;
			ELSIF tmr01.q THEN
				step := step + 10000;
			END_IF
			
		END_IF	
		
	202:
		bdone := TRUE;
		step := 0;
	
		
		
END_CASE
END_ACTION

ACTION tmrAct:
tmr01();
END_ACTION

METHOD Up : BOOL
VAR_INPUT
	// 動作的台車 bit0:台車1、bit0:台車2、bit0:台車3、bit0:台車4
	Action_Select : WORD := 0;
END_VAR
IF Action_Select = 0 THEN
	Module_Select := 255;
ELSE
	Module_Select := Action_Select;
END_IF
	
step := 100;
END_METHOD

END_PROGRAM

// ---- POUs/硬體控制/AxisAction.TcPOU
PROGRAM AxisAction
VAR
	bBoot : BOOL := true;

	bMove: BOOL;
	tof_PowerOff: TOF;
	ldf_PowerOff: F_TRIG;
END_VAR

IF bBoot THEN
	initAction();
	bBoot := FALSE;
END_IF



Axis.FeedCar();

METHOD initAction : BOOL
VAR_INPUT
END_VAR
FeedCar.Encoder := ADR(axis.FeedCar_Enc);

FeedCar.Set_VFD_IO(
	FWD:= ADR(io.q104), 
	REV:= ADR(io.q105), 
	Speed_Io_1:= ADR(io.q106), 
	Speed_Io_2:= ADR(io.q107), 
	Speed_Io_3:= ADR(io.q108), 
	Reset:= ADR(io.q307), 
	Run:= ADR(io.i107), 
	Error:= ADR(io.i108)
);

FeedCar.SetLimit_IO(
	Origin:= ADR(io.i213), 
	P_Limit:= 0, 
	N_Limit:= 0
);

FeedCar.Name := "FeedCar";
END_METHOD

END_PROGRAM

// ---- POUs/動作流程控制/FeedMain.TcPOU
PROGRAM FeedMain
VAR
	step: UINT;
	
	tmr01: TON;
	tmr8000: TON;
	
	tmr_ErrorReset: TON;
	
	
	// 註冊料總寬度
	Wide_Size : LREAL;
	
	// 容許誤差
	Wide_Max : LREAL;
	Wide_Min : LREAL;
	// 進料寬度檢測通過
	Wide_Check_Pass : BOOL;
	// 進料數量
	inputNumber : int;
	
	// 分料位置 計算結果 (有分料的起始位置 與 分料的停止位置)
	AlignmentPosArr : ARRAY [0..10] OF Alignment_pos;
	// 分料數量
	AlignmentCount : INT; 
	
	
	// 投料搬移 搬移次數
	feed_MoveCycle: DINT;
	// 投料搬移 起始距離
	feed_MoveStartPos: LREAL; 
	// 投料搬移 最後一次位置
	feed_MoveLastPos: LREAL;
	
	// 進料數量
	FeedNumber : INT;
	
	// 已就緒
	bReady : BOOL;
	
	i1: INT;
	i2: INT;
	dint_tmp1 : DINT;
	dint_tmp2 : DINT;
	lreal_tmp1 : LREAL;
	
	// 台車位置紀錄
	Jog_car_at : INT;
	// 啟動的模式
	StartMode: INT;
	
	StrMem : WStrMem;
	
	
	_log : Step_Log; 
END_VAR

VAR_OUTPUT
	bBuzy: BOOL;
	bError: BOOL;
	bDone: BOOL;
	iErrorId : DINT;
END_VAR

VAR RETAIN PERSISTENT
	// 輸入的寬度暫存 (防止運作中輸入質發生變動)
	Workpiece_Width_array_tmp: ARRAY [0..10] OF LREAL;
END_VAR

IF (EStop OR SystemError OR Input.Feed_Reset) AND bBuzy THEN
	IF bBuzy THEN
		step := step  + 10000;
	END_IF
END_IF

bBuzy := (step >= 1 AND step <> 806 AND step < 10000);
bError := (step >= 10000);

// tmr_ErrorReset(in:= bError, PT:=T#1S);
// IF tmr_ErrorReset.Q THEN
// 	iErrorId := step - 10000;
// 	step := 0;
// END_IF

IF (Safety.SystemError) AND bError THEN
	bReady := FALSE;
END_IF

IF step <> 0 AND Feed_Reset THEN
	iErrorId := step - 10000;
	step := 0;
END_IF

IF Input.Feed_Start AND (step > 10000 OR  Safety.SystemError) THEN
	Safety.SystemError := FALSE;
	step := 0;
END_IF

IF Pause THEN
	RETURN;
END_IF

Step_0_Main();


Timer();

Output.ActionMode_Now := step;

Output.in_Pos_sensor := 0;
Output.in_Pos_sensor.0 := IO.i402;
Output.in_Pos_sensor.1 := IO.i404;
Output.in_Pos_sensor.2 := IO.i406;
Output.in_Pos_sensor.3 := IO.i408;

Output.Out_Pos_sensor := 0;

Output.Out_Pos_sensor.0 := IO.i113;
Output.Out_Pos_sensor.1 := IO.i114;
Output.Out_Pos_sensor.2 := IO.i115;

_log(name := 'FeedMain', step := step);

// 計算分料的起始位置
METHOD INTERNAL Alignment_End_Pos : LREAL


VAR_INPUT
	NumberOfArray : INT;
END_VAR

VAR
	i : INT;
	tmp1 : LREAL;
	tmp2 : LREAL;
	tmp3 : LREAL;
	tmp4 : LREAL;
END_VAR
// 第二支料分離結束位置 =  工件待命位置 + 臺車寬度 - (第一支料寬 + 第二支料寬 + 材料排列間距)

// 工件待命位置 + 臺車寬度
tmp1 := Config.pos_Workpiace_StanbyPoint + Config.FeedCar_Length;

// 輸入不為0時
IF NumberOfArray >= 0 THEN
	tmp2 := 0;

	IF NumberOfArray > 0 THEN
		FOR i := 0 TO NumberOfArray - 1 DO
			// 料寬 + 材料排列間距 的累計
			tmp2 := tmp2 + Workpiece_Width_array_tmp[i] + Config.dis_Alignment;
		END_FOR
	END_IF
	
	tmp3 := Workpiece_Width_array_tmp[NumberOfArray];
	
	tmp4 := tmp1 - (tmp2 + tmp3);
ELSE
	tmp4 := 0;
END_IF

Alignment_End_Pos := tmp4;
END_METHOD

// 計算分料的起始位置
METHOD INTERNAL Alignment_Start_Pos : LREAL


VAR_INPUT
	NumberOfArray : INT;
END_VAR

VAR
	i : INT;
	tmp1 : LREAL;
	tmp2 : LREAL;
	tmp3 : LREAL;
	tmp4 : LREAL;
END_VAR
// 工件待命位置 + 臺車寬度
tmp1 := Config.pos_Workpiace_StanbyPoint + Config.FeedCar_Length;

// 輸入不為0時
IF NumberOfArray >= 0 THEN
	tmp2 := 0;
	
	IF NumberOfArray > 0 THEN
		FOR i := 0 TO NumberOfArray - 1 DO
			// 料寬累計
			tmp2 := tmp2 + Workpiece_Width_array_tmp[i];
		END_FOR
	END_IF
	
	tmp3 := (Workpiece_Width_array_tmp[NumberOfArray] / 2);
	
	tmp4 := tmp1 - (tmp2 + tmp3);
	
ELSE
	
	tmp4 := 0;
	
END_IF

Alignment_Start_Pos := tmp4;
END_METHOD

// 計算分料的起始位置
METHOD INTERNAL Feed_Start_Pos : LREAL


VAR_INPUT
	NumberOfArray : INT;
END_VAR

VAR
	i : INT;
	tmp1 : LREAL;
	tmp2 : LREAL;
	tmp3 : LREAL;
	tmp4 : LREAL;
END_VAR
// 第一支進料移動起始位置 =  工件待命位置 + 臺車寬度 - (第一支料寬 + 材料排列間距)

// 工件待命位置 + 臺車寬度
tmp1 := Config.pos_Workpiace_StanbyPoint + Config.FeedCar_Length;

FOR i := 0 TO NumberOfArray - 1 DO
	// // 料寬 + 材料排列間距 的累計
	tmp2 := tmp2 + Workpiece_Width_array_tmp[i] + Config.dis_Alignment;
END_FOR

tmp3 := Workpiece_Width_array_tmp[i] + (Config.dis_Alignment / 2);

tmp4 := tmp1 - (tmp2 + tmp3);

Feed_Start_Pos := tmp4;
END_METHOD

ACTION Step_0_Main:
(*======================================
		確認起動條件&回原點
  ======================================*)

// 處裡緊急停止訊號

output.Feed_bBuzy := bbuzy;
output.Feed_bdone := bdone;
Output.Feed_bError := bError;
Output.Feed_Workpiace_H := Sensor.MeasureValue;
Output.Feed_Workpiace_W := HeightMeasurer.MeasureValue;

step_0100_Homming();
step_0400_input();
step_0600_Alignment();
step_0800_Feeding();
step_1000_DB_Data_Change();
step_2000_Push_site();

step_3400_input_WeightError();
Step_8000_Jog_Start();

CASE step OF
	0:
		IF Input.Feed_Start THEN
			step := 1;
			StartMode := Input.Feed_Mode;
		END_IF
		
	
	1:
		bDone := FALSE;
		IF StartMode = 8000 THEN
			step := 8000;
		ELSIF StartMode = 8001 THEN
			step := 0;
		ELSIF StartMode = 2000 THEN
			step := 2000;
		ELSE
			step := step + 1;
		END_IF
		
	2: // 沒就緒狀態，先歸零
		IF NOT bReady OR StartMode = 100 THEN
			step := 100;
		ELSE
			step := step + 1;
		END_IF
		
	3:
		step := 10;
		
(*	================================
			從資料庫取得資料
	================================	*)
	10:
		ReadSQLData.Get_WorkkOrder();
		step := step + 1;
		
	11:
		IF ReadSQLData.bBuzy OR ReadSQLData.bError THEN
			step := step + 1;
		END_IF
		
	12:
		IF ReadSQLData.bDone THEN
			step := step + 1;
		ELSIF ReadSQLData.bError THEN
			step := step + 10000;
		END_IF
		
	13:
		step := 20;
		
(*	================================
			確認要執行的動作
	================================	*)
	20: // 檢查待命區是否還有料
		IF ProjectData.WorkOrder_Nunber_At_waitLoading > 0 THEN
			step := 800;
		ELSIF ProjectData.WorkOrder_Nunber_At_holding > 0 THEN
			step := 400;
		ELSE
			pMsg.Push_Alarm_NoPause(STR := WStrConcat(
				"FeedMain:沒有狀態是 暫存中(holding)　或　等待上料(waitLoading) 的料(",
				TO_WSTRING(step),
				")"
			));
			bDone := TRUE;
			step := 0;
		END_IF
	
		
END_CASE
END_ACTION

ACTION step_0100_Homming:
CASE step OF
	100:// 復歸定位圓柱、台車升降、測高
		Hydraulic.CarLift_Down(0);
		StopPin.Down(0);
		HeightMeasurer.Homing();
		step := step + 1;
		
	101:
		IF (Hydraulic.bBuzy OR Hydraulic.bError) AND (StopPin.bBuzy OR StopPin.bError)
			AND (HeightMeasurer.bBuzy OR HeightMeasurer.bError) THEN
			step := step + 1;
		END_IF
		
	102:
		IF Hydraulic.bDone THEN
			step := step + 1;
		ELSIF Hydraulic.bError THEN
			step := step + 10000;
		END_IF
		
	103:
		step := 110;
	
	110:
		IF FeedCar.bHome AND StartMode = 0 THEN
			step := step + 10;
		ELSE
			step := step + 1;
		END_IF
		
	111:
		FeedCar.Homing();
		step := step + 1;
		
	112:
		IF (FeedCar.bBuzy OR FeedCar.bError) THEN
			step := step + 1;
		END_IF
		
	113:
		IF FeedCar.bDone THEN
			step := step + 1;
		ELSIF FeedCar.bError THEN
			step := step + 10000;
		END_IF
		
	114:
		step := 120;
		
	120:
		FeedCar.AbsMove(0,0);
		step := step + 1;
		
	121:
		IF (FeedCar.bBuzy OR FeedCar.bError) THEN
			step := step + 1;
		END_IF
		
	122:
		IF FeedCar.bDone AND StopPin.bDone AND HeightMeasurer.bDone THEN
			step := step + 1;
		ELSIF FeedCar.bError THEN
			step := step + 10000;
		END_IF
		
	123:
		step := 130;
		
	130:
		FeedCar.AbsMove(config.pos_StartPoint, 0);
		step := step + 1;
		
	131:
		IF (FeedCar.bBuzy OR FeedCar.bError) THEN
			step := step + 1;
		END_IF
		
	132:
		IF FeedCar.bDone THEN
			step := step + 1;
		ELSIF FeedCar.bError THEN
			step := step + 10000;
		END_IF
		
	133:
		step := 140;
		
	140:
		bReady := TRUE;
		step := step + 1;
		
	141:
		IF StartMode = 0 THEN
			step := 10;
		ELSE
			bDone := TRUE;
			step := 0;
		END_IF
		
END_CASE
END_ACTION

ACTION step_0400_input:
CASE step OF
(*	============================================
			從資料庫取得吊掛區的註冊工件
	============================================*)
	400:
		step := step + 1;
		
	401:
		ReadSQLData.Get_WorkkOrder();
		step := step + 1;
		
	402:
		IF ReadSQLData.bBuzy OR ReadSQLData.bError THEN
			step := step + 1;
		END_IF
		
	403:
		IF ReadSQLData.bDone THEN
			step := step + 1;
		ELSIF ReadSQLData.bError THEN
			step := step + 10000;
		END_IF

	404:
		IF ProjectData.WorkOrder_Nunber_At_waitLoading > 0 THEN
 			step := 790;
		ELSIF ProjectData.WorkOrder_Nunber_At_holding > 0 THEN
			step := step + 1;
		ELSE
			pMsg.Push_Alarm_NoPause(STR := WStrConcat(
				"FeedMain:沒有狀態是 暫存中(holding) 的料(",
				TO_WSTRING(step),
				")"
			));
			step := 0;
		END_IF

	405:
		step := 410;
			
		
(*	============================================
					計算總寬度
	============================================*)
	410: // 資料初始化				
		FOR i1 := 0 TO 10 DO
			Workpiece_Width_array_tmp[i1] := ProjectData.WorkOrder_At_holding[i1].Height;
		END_FOR
		
		Wide_Size := 0;
		step := step + 1;
		
	411: // 加總所有吊掛區的工件寬度
		FOR i1 := 0 TO ProjectData.WorkOrder_Nunber_At_holding - 1 DO
			Wide_Size := Wide_Size + Workpiece_Width_array_tmp[i1];
		END_FOR
		step := step + 1;
		
	412:
		step := 420;

(*	============================================
			開始整直 與 驗證註冊資料是否正確
	============================================*)
	420:// 臺車下降、定位圓柱升起
		Hydraulic.CarLift_Down();
		StopPin.up();
		step := step + 1;
		
	421:
		IF (Hydraulic.bBuzy OR Hydraulic.bError) AND (StopPin.bBuzy OR StopPin.bError) THEN
			step := step + 1;
		END_IF
		
	422:
		IF Hydraulic.bDone AND StopPin.bDone THEN
			step := step + 1;
		ELSIF Hydraulic.bError OR StopPin.bError THEN
			step := step + 10000;
		END_IF
		
	423:
		step := 430;
		
	430: // 臺車 移動到 搬移起始點
		FeedCar.AbsMove(0);
		step := step + 1;
		
	431:
		IF (FeedCar.bBuzy OR FeedCar.bError) THEN
			step := step + 1;
		END_IF
		
	432:
		IF FeedCar.bDone THEN
			step := step + 1;
		ELSIF FeedCar.bError THEN
			step := step + 10000;
		END_IF
		
	433:
		step := 440;
		
	440:// 臺車 上升到中位
		Hydraulic.CarLift_Mid();
		step := step + 1;
		
	441:
		IF (Hydraulic.bBuzy OR Hydraulic.bError) THEN
			step := step + 1;
		END_IF
		
	442:
		IF Hydraulic.bDone THEN
			step := step + 1;
		ELSIF Hydraulic.bError THEN
			pMsg.Push_Alarm_NoPause(STR := WStrConcat(
				"FeedMain:執行整料動作時發生錯誤(",
				TO_WSTRING(step),
				")"
			));
		END_IF
		
	443:
		step := 450;
		
	450:// 臺車 做寬度測量
		FeedCar.Find();
		step := step + 1;
		
	451:
		IF (FeedCar.bBuzy OR FeedCar.bError) THEN
			step := step + 1;
		END_IF
		
	452:
		IF FeedCar.bDone THEN
			step := step + 1;
		ELSIF FeedCar.bError THEN
			step := step + 10000;
		END_IF
		
	453: // 驗證註冊資料
		Wide_Check_Pass := FALSE;
		// 誤差上限
		Wide_Max := Wide_Size + (Wide_Size * config.Workpiace_Err_size);
		// 誤差下限
		Wide_Min := Wide_Size - (Wide_Size * config.Workpiace_Err_size);
		
		// 判斷寬度是否在誤差範圍內
		Wide_Check_Pass := Wide_Min < FeedCar.rFindPos AND Wide_Max > FeedCar.rFindPos;
		
		step := step + 1;
		
	454:
		step := 460;
		
	460:// 臺車下降，定位圓柱下降
		StopPin.Down();
		step := step + 1;
		
	461:
		IF (StopPin.bBuzy OR StopPin.bError) THEN
			step := step + 1;
		END_IF
		
	462:
		step := 470;
		
	470:
		IF Wide_Check_Pass THEN
			// 通過寬度檢測
			step := step + 1;
		ELSE
			// 寬度檢測失敗
			step := 3400;
		END_IF
		
	471:
		step := 480;
	
	480:
		FeedCar.AbsMove(config.pos_StartPoint, 1);
		step := step + 1;
		
	481:
		IF (FeedCar.bBuzy OR FeedCar.bError) THEN
			step := step + 1;
		END_IF
		
	482:
		IF FeedCar.bDone THEN
			step := step + 1;
		ELSIF FeedCar.bError THEN
			step := step + 10000;
		END_IF
		
	483:
		step := 490;
		
	490:
		Hydraulic.CarLift_Up(0);
		step := step + 1;
		
	491:
		IF (Hydraulic.bBuzy OR Hydraulic.bError) THEN
			step := step + 1;
		END_IF
		
	492:
		IF Hydraulic.bDone THEN
			step := step + 1;
		ELSIF Hydraulic.bError THEN
			step := step + 10000;
		END_IF
		
	493:
		FeedCar.AbsMove(FeedCar.Pos - 10);
		step := step + 1;
		
	494:
		IF (FeedCar.bBuzy OR FeedCar.bError) THEN
			step := step + 1;
		END_IF
		
	495:
		IF FeedCar.bDone AND StopPin.bDone THEN
			step := step + 1;
		ELSIF FeedCar.bError OR StopPin.bError THEN
			step := step + 10000;
		END_IF
		
	496:
		step := 500;
		
	500: // 判斷是否有只有一隻料，只有一支料直接送入進料區
		IF ProjectData.WorkOrder_Nunber_At_waitLoading = 0 AND ProjectData.WorkOrder_Nunber_At_holding = 1 AND	// 只有一支料
			(Feed_Enable AND NOT IO.i402 AND NOT IO.i404) THEN 													// 允許進料狀態
 			step := 550;
		ELSE
			step := step + 1;
		END_IF	
		
		
(*	================== 標準進料流程 ==================*)		
	501:
		FeedCar.AbsMove(config.pos_Workpiace_StanbyPoint, 1);
		step := step + 1;
		
	502:
		IF (FeedCar.bBuzy OR FeedCar.bError) THEN
			step := step + 1;
		END_IF
		
	503:
		IF FeedCar.bDone THEN
			step := step + 1;
		ELSIF FeedCar.bError THEN
			step := step + 10000;
		END_IF
		
	504:
		step := 510;
		
	510: // 臺車下降
		Hydraulic.CarLift_Down();
		step := step + 1;
		
	511:
		IF (Hydraulic.bBuzy OR Hydraulic.bError) THEN
			step := step + 1;
		END_IF
		
	512:
		IF Hydraulic.bDone THEN
			step := step + 1;
		ELSIF Hydraulic.bError THEN
			step := step + 10000;
		END_IF
		
	513:
		step := 600;
		
(*	================== 只進一支料流程 ==================*)
	550:
		ReadSQLData.Set_Work_Order_Status( 
			uuid := ProjectData.WorkOrder_At_holding[0].steel_id,
			status := 'inSide',
			location := 'entranceRack'
			);
		step := step + 1;
		
	551:
		IF ReadSQLData.bBuzy OR ReadSQLData.bError THEN
			step := step + 1;
		END_IF
		
	552:
		IF ReadSQLData.bDone THEN
			step := step + 1;
		ELSIF ReadSQLData.bError THEN
			step := step + 10000;
		END_IF
		
	553:
		step := 900;
END_CASE
END_ACTION

ACTION step_0600_Alignment:
(*
	1.取出
*)

CASE step OF
	600: // 判斷是否需要執行分料動作
		inputNumber := TO_INT(ProjectData.WorkOrder_Nunber_At_holding);
		IF inputNumber > 1 THEN
			step := step + 1;
		ELSE
			step := 700; 
		END_IF
		
	601: // 計算分隔距離與台車移動的距離
		FOR i1 := 0 TO 10 DO
			IF i1 <= inputNumber THEN
				AlignmentPosArr[i1].Start := Alignment_Start_Pos(i1);
				AlignmentPosArr[i1].End := Alignment_End_Pos(i1);
			ELSE
				AlignmentPosArr[i1].Start := 0;
				AlignmentPosArr[i1].End := 0;
			END_IF
		END_FOR
		step := step + 1;
		
	602:
		i2 := inputNumber - 1;
		step := step + 1;
		
	603:
		step := 610;
		
	610: // 臺車 移動到 材料 分離起始位置
		FeedCar.AbsMove(AlignmentPosArr[i2].Start, 1);
		step := step + 1;
		
	611:
		IF (FeedCar.bBuzy OR FeedCar.bError) THEN
			step := step + 1;
		END_IF
		
	612:
		IF FeedCar.bDone THEN
			step := step + 1;
		ELSIF FeedCar.bError THEN
			step := step + 10000;
		END_IF
		
	613:
		step := 620;
		
	620: // 台車 升到 中位
		Hydraulic.CarLift_Mid(0);
		step := step + 1;
		
	621:
		IF (Hydraulic.bBuzy OR Hydraulic.bError) THEN
			step := step + 1;
		END_IF
		
	622:
		IF Hydraulic.bDone THEN
			step := step + 1;
		ELSIF Hydraulic.bError THEN
			step := step + 10000;
		END_IF
		
	623:
		step := 630;
		
	630: // 臺車 移動到 材料分離位置
		FeedCar.AbsMove(AlignmentPosArr[i2].End, 0);
		step := step + 1;
		
	631:
		IF (FeedCar.bBuzy OR FeedCar.bError) THEN
			step := step + 1;
		END_IF
		
	632:
		IF FeedCar.bDone THEN
			step := step + 1;
		ELSIF FeedCar.bError THEN
			step := step + 10000;
		END_IF
		
	633:
		step := 640;
		
	640: // 台車 降到 低位
		Hydraulic.CarLift_Down(0);
		step := step + 1;
		
	641:
		IF (Hydraulic.bBuzy OR Hydraulic.bError) THEN
			step := step + 1;
		END_IF
		
	642:
		IF Hydraulic.bDone THEN
			step := step + 1;
		ELSIF Hydraulic.bError THEN
			step := step + 10000;
		END_IF
		
	643:
		step := 650;
		
	650:
		// 待分離數量 -1
		i2 := i2 - 1;
		IF i2 > 0 THEN
			step := 610;
// 			step := 652;
		ELSE
			step := step + 1;
		END_IF
		
	651:// 歸零已給料數量
		step := 700;
		
		
	700:
		FeedNumber := 0;
		i1 := 0;
		step := step + 1;
		
	701:
		// 將放置(搬移起始)位置寫入資料庫
		ReadSQLData.Set_Work_Order_WaitLoading_Pos( 
			id := i1,
			Pos := Feed_Start_Pos(i1)
			);
		step := step + 1;
		
	702:
		IF ReadSQLData.bBuzy OR ReadSQLData.bError THEN
			step := step + 1;
		END_IF
		
	703:
		IF ReadSQLData.bDone THEN
			step := step + 1;
		ELSIF ReadSQLData.bError THEN
			step := step + 10000;
		END_IF
		
	704:
		i1 := i1 + 1;
		IF i1 < ProjectData.WorkOrder_Nunber_At_holding THEN
			step := 701;
		ELSE
			step := step + 1;
		END_IF
		
	705:
		step := 710;
		
	710:
		// 將放置(搬移起始)位置寫入資料庫
		ReadSQLData.Get_WorkkOrder();
		step := step + 1;
		
	711:
		IF ReadSQLData.bBuzy OR ReadSQLData.bError THEN
			step := step + 1;
		END_IF
		
	712:
		IF ReadSQLData.bDone THEN
			step := step + 1;
		ELSIF ReadSQLData.bError THEN
			step := step + 10000;
		END_IF
		
	713:
		tmr01.PT := T#500MS;
		tmr01.IN := TRUE;
		IF tmr01.Q THEN
			tmr01.IN := FALSE;
			step := step + 1;
		END_IF
		
	714:
		step := 790;
		
	
	790:
		i2 := 0;
		step := step + 1;
		
	791:
		ReadSQLData.Set_Work_Order_2_waitLoading(i2);
		step := step + 1;
		
	792:
		IF ReadSQLData.bBuzy OR ReadSQLData.bError THEN
			step := step + 1;
		END_IF
		
	793:
		IF ReadSQLData.bDone OR ReadSQLData.bError THEN
			step := step + 1;
		END_IF
		
	794:
		i2 := i2 + 1;
		IF i2 < ProjectData.WorkOrder_Nunber_At_holding THEN 
			step := 791;
		ELSE
			step := 795;
		END_IF 
		
		
	795:
		step := 800;
		
END_CASE
END_ACTION

ACTION step_0800_Feeding:
CASE step OF
	800:
		ReadSQLData.Get_WorkkOrder();
		step := step + 1;
		
	801:
		IF ReadSQLData.bBuzy OR ReadSQLData.bError THEN
			step := step + 1;
		END_IF
		
	802:
		IF ReadSQLData.bDone THEN
			step := step + 1;
		ELSIF ReadSQLData.bError THEN
			step := step + 10000;
		END_IF
		
	803:
		tmr01.PT := T#500MS;
		tmr01.IN := TRUE;
		IF tmr01.Q THEN
			tmr01.IN := FALSE;
			step := step + 1;
		END_IF
		
		
	804: // 確定有等待進料的料
		IF  ProjectData.WorkOrder_Nunber_At_waitLoading > 0 THEN
			step := step + 1;
		ELSE
			IF ProjectData.WorkOrder_Nunber_At_waitLoading <= 0 THEN
				// 等待投料位置的原料數為0
				pMsg.Push_Error(WStrConcat(
					"FeedMain: 等待投料位置的原料數為0"
					));
			ELSE
				// 有料正在加工中
				pMsg.Push_Error(WStrConcat(
					"FeedMain: 有料正在加工中"
					));
			END_IF
			step := step + 10000;
		END_IF
		
		
		
	805: // 檢查等待進料的料位置是否正確
		IF ProjectData.WorkOrder_At_waitLoading[0].waitLoading_pos > Config.pos_CarPin_StopPoint AND	// 位置大於 定位PIN()
			ProjectData.WorkOrder_At_waitLoading[0].waitLoading_pos < Config.pos_Workpiace_FeedPoint THEN	// 位置小於 投料位置(2700) - 台車平台大小(1080)
			step := step + 1;
		ELSE
			pMsg.Push_Error(WStrConcat(
				"FeedMain: ",
				WLEFT(STR:= TO_WSTRING(ProjectData.WorkOrder_At_waitLoading[0].steel_id), SIZE:= 8),
				" :的待命位置錯誤: ",
				TO_WSTRING(ProjectData.WorkOrder_At_waitLoading[0].waitLoading_pos)
				));
			step := step + 10000;
		END_IF
		
	806:
		IF Feed_Enable AND NOT IO.i402 AND NOT IO.i404 THEN
			step := 810;
		END_IF
		

	810: 
		step := step + 1;
		
	811: // 計算搬移次數
		// 料移動起始位置
		dint_tmp1 := TO_DINT(ProjectData.WorkOrder_At_waitLoading[0].waitLoading_pos);
		
		// 移動距離 = 投料位置 - 第一支進料移動起始位置
		dint_tmp2 := TO_DINT( config.pos_Workpiace_FeedPoint) - dint_tmp1;
		
		IF dint_tmp2 > 0 THEN // 當可移動距離 < 台車寬度
			lreal_tmp1 := (config.FeedCar_Length - (ProjectData.WorkOrder_At_waitLoading[0].Height + 50)) / dint_tmp2;
			
			IF lreal_tmp1 >= 1 THEN
				feed_MoveCycle := TO_INT(TO_STRING(lreal_tmp1));
			ELSE
				feed_MoveCycle := 0;
			END_IF
			
			feed_MoveStartPos := dint_tmp1;		// 次數內的 搬移起始位置
			
			// 最後一次的搬移起始位置
			feed_MoveLastPos := config.pos_Workpiace_FeedPoint - 
									(Config.FeedCar_Length - (ProjectData.WorkOrder_At_waitLoading[0].Height + 50)) +
									(dint_tmp2 * feed_MoveCycle);
			
			step := step + 1;
		ELSE // 當可移動距離 > 台車寬度
			
			// 重複移動次數 0
			feed_MoveCycle := 0; 
			// 搬移 起始位置
			feed_MoveStartPos := dint_tmp1;
			// 最後一次的搬移 起始位置 = 投料位置 - (臺車寬度 - (工件寬度 + 50))
			feed_MoveLastPos := config.pos_Workpiace_FeedPoint - 
									(Config.FeedCar_Length - (ProjectData.WorkOrder_At_waitLoading[0].Height + 50));
			step := step + 1;
		END_IF
		
	812:
		IF NOT HeightMeasurer.bBuzy THEN
			IF NOT io.i314 THEN
				// 測高機構不再原點，會導致撞機
				step := step + 10000;
			ELSE
				step := step + 1;
			END_IF
		END_IF
		
	813:
		step := 820;
		
		
	820: // 降下台車
		Hydraulic.CarLift_Down(0);
		step := step + 1;
		
	821:
		IF (Hydraulic.bBuzy OR Hydraulic.bError) THEN
			step := step + 1;
		END_IF
		
	822:
		IF Hydraulic.bDone THEN
			step := step + 1;
		ELSIF Hydraulic.bError THEN
			step := step + 10000;
		END_IF
		
	823:
		step := 830;
		
	830: // 臺車 移動到 搬移起始點
		step := step + 1;
	831:
		FeedCar.AbsMove(feed_MoveStartPos,1);
		step := step + 1;
		
	832:
		IF (FeedCar.bBuzy OR FeedCar.bError) THEN
			step := step + 1;
		END_IF
		
	833:
		IF FeedCar.bDone THEN
			step := step + 1;
		ELSIF FeedCar.bError THEN
			step := step + 10000;
		END_IF
		
	834:
		step := 840;
		
	840: // 上升台車
		Hydraulic.CarLift_Up(0);
		step := step + 1;
		
	841:
		IF (Hydraulic.bBuzy OR Hydraulic.bError) THEN
			step := step + 1;
		END_IF
		
	842:
		IF Hydraulic.bDone THEN
			step := step + 1;
		ELSIF Hydraulic.bError THEN
			step := step + 10000;
		END_IF
		
	843:
		step := 850;
		
	850: // 臺車 移動到 投料輸送機 位置
		FeedCar.AbsMove(config.pos_Workpiace_FeedPoint,1);
		step := step + 1;
		
	851:
		IF (FeedCar.bBuzy OR FeedCar.bError) THEN
			step := step + 1;
		END_IF
		
	852:
		IF FeedCar.bDone THEN
			step := step + 1;
		ELSIF FeedCar.bError THEN
			step := step + 10000;
		END_IF
		
	853:
		step := 860;
		
	860: // 臺車下降
		Hydraulic.CarLift_Down(0);
		step := step + 1;
		
	861:
		IF (Hydraulic.bBuzy OR Hydraulic.bError) THEN
			step := step + 1;
		END_IF
		
	862:
		IF Hydraulic.bDone THEN
			step := step + 1;	
		ELSIF Hydraulic.bError THEN
			step := step + 10000;
		END_IF
		
	863:
		step := 870;
		
	870: // 搬移次數 -1 後，判斷搬移次數是否大於1 大於 -> 繼續完整搬移 小於 -> 使用最後位置搬移
		
		IF feed_MoveCycle > 0 THEN
			feed_MoveCycle := feed_MoveCycle - 1;
			step := 830;
		ELSE
			step := 880;
		END_IF
			
			
	880:
		IF feed_MoveLastPos + 100 > config.pos_Workpiace_FeedPoint THEN
			step := 910;
		ELSE
			step := step + 1;
		END_IF
		
	881: // 一到最後一次的 開始搬移位置
		FeedCar.AbsMove(feed_MoveLastPos,1);
		step := step + 1;
		
	882: // 
		IF (FeedCar.bBuzy OR FeedCar.bError) THEN
			step := step + 1;
		END_IF
		
	883:
		IF FeedCar.bDone THEN
			step := step + 1;
		ELSIF FeedCar.bError THEN
			step := step + 10000;
		END_IF
		
	884:
		step := 890;
	
	890: // 臺車上升
		Hydraulic.CarLift_Up(0);
		step := step + 1;
		
	891:
		IF (Hydraulic.bBuzy OR Hydraulic.bError) THEN
			step := step + 1;
		END_IF
		
	892:
		IF Hydraulic.bDone THEN
			step := step + 1;
		ELSIF Hydraulic.bError THEN
			step := step + 10000;
		END_IF
		
	893:
		step := 900;
		
	900: // 臺車 移動到 投料輸送機 位置
		FeedCar.AbsMove(config.pos_Workpiace_FeedPoint,1);
		step := step + 1;
		
	901:
		IF (FeedCar.bBuzy OR FeedCar.bError) THEN
			step := step + 1;
		END_IF
		
	902:
		IF FeedCar.bDone THEN
			step := step + 1;
		ELSIF FeedCar.bError THEN
			step := step + 10000;
		END_IF
		
	903:
		step := 910;
		
		
	910: // 降下台車
		Hydraulic.CarLift_Down(0);
		step := step + 1;
		
	911:
		IF (Hydraulic.bBuzy OR Hydraulic.bError) THEN
			step := step + 1;
		END_IF
		
	912:
		IF Hydraulic.bDone THEN
			step := step + 1;
		ELSIF Hydraulic.bError THEN
			step := step + 10000;
		END_IF
		
	913:
		step := 1000;
END_CASE
END_ACTION

ACTION step_1000_DB_Data_Change:
CASE step OF
	1000:
		ReadSQLData.Set_Work_Order_2_inSide(0);
		step := step + 1;
		
		
	1001:
		IF ReadSQLData.bBuzy OR ReadSQLData.bError THEN
			step := step + 1;
		END_IF
		
	1002:
		IF ReadSQLData.bDone THEN 
			step := step + 1;
		ELSIF ReadSQLData.bError THEN
			step := step + 10000;
		END_IF
		
	1003:
		step := 1010;

		
	1010: // 給料靠邊、台車移到下一支材料位置 或 回進料點
		PullOver.Start();
		step := step + 1;
		
	1011:
		IF (PullOver.bBuzy OR PullOver.bError) THEN
			step := step + 1;
		END_IF
		
	1012:
		step := 1020;
		
	1020:
		ReadSQLData.Get_WorkkOrder();
		step := step + 1;
		
		
	1021:
		IF ReadSQLData.bBuzy OR ReadSQLData.bError THEN
			step := step + 1;
		END_IF
		
	1022:
		IF ReadSQLData.bDone THEN 
			step := step + 1;
		ELSIF ReadSQLData.bError THEN
			step := step + 10000;
		END_IF
		
	1023:
		step := 1030;
		
		
	1030:
		IF ProjectData.WorkOrder_Nunber_At_waitLoading > 0 THEN
			// 還有 等待進料狀(waitLoading) 的料的
			FeedCar.AbsMove(ProjectData.WorkOrder_At_waitLoading[0].waitLoading_pos ,1);
		ELSE
			// 所有 等待進料(waitLoading) 的料都已完成
			FeedCar.AbsMove(config.pos_StartPoint,1);
		END_IF
		step := step + 1;
		
	1031:
		IF(FeedCar.bBuzy OR FeedCar.bError) THEN
			step := step + 1;
		END_IF
		
	1032:
		IF PullOver.bDone THEN
			step := step + 1;
		ELSIF PullOver.bError OR FeedCar.bError THEN
			step := step + 10000;
		END_IF
		
	1033:
		step := 1040;
		
	1040:
		ReadSQLData.Get_WorkkOrder();
		step := step + 1;
		
	1041:
		IF ReadSQLData.bBuzy OR ReadSQLData.bError THEN
			step := step + 1;
		END_IF
		
	1042:
		IF ReadSQLData.bDone THEN
			step := step + 1;
		ELSIF ReadSQLData.bError THEN
			step := step + 10000;
		END_IF
		
	1043:
		step := 1050;
		
	
	1050:
		bDone := TRUE;
		step := step + 1;
		
	1051:
		tmr01.PT := T#500MS;
		tmr01.IN := TRUE;
		IF tmr01.Q THEN
			tmr01.IN := FALSE;
			step := step + 1;
		END_IF
		
	1052:
		IF ProjectData.WorkOrder_Nunber_At_waitLoading > 0 THEN
			step := 800;
		ELSIF ProjectData.WorkOrder_Nunber_At_holding <= 0 THEN
			step := 0;
		ELSE
			StartMode := 400;
			step := 400;
		END_IF
		
END_CASE
END_ACTION

ACTION step_2000_Push_site:
CASE step OF
	2000: // 給料靠邊、台車移到下一支材料位置 或 回進料點
		bDone := FALSE;
		Hydraulic.Over_Pull(0);
		step := step + 1;
		
	2001:
		IF (Hydraulic.bBuzy1 OR Hydraulic.bError1) THEN
			step := step + 1;
		END_IF
		
	2002:
		IF Hydraulic.bDone1 THEN
			step := step + 1;
		ELSIF Hydraulic.bError1 THEN
			step := step + 10000;
		END_IF
		
	2003:
		step := 2010;
		
	2010:
		HeightMeasurer.Measure();
		step := step + 1;
		
	2011:
		IF (HeightMeasurer.bBuzy OR HeightMeasurer.bError) THEN
			step := step + 1;
		END_IF
		
	2012:
		IF HeightMeasurer.bDone THEN
			step := step + 1;
		ELSIF HeightMeasurer.bError THEN
			step := step + 10000;
		END_IF
		
	2013:
		step := 2020;
		
	
	2020:
		bDone := TRUE;
		step := 0;
		
END_CASE
END_ACTION

ACTION step_3400_input_WeightError:
CASE step OF
	3400:
		Hydraulic.CarLift_Up(0);
		step := step + 1;
		
	3401:
		IF (Hydraulic.bBuzy OR Hydraulic.bError) THEN
			step := step + 1;
		END_IF
		
	3402:
		IF Hydraulic.bDone THEN
			step := step + 1;
		ELSIF Hydraulic.bError THEN
			step := step + 10000;
		END_IF
		
	3403:
		step := 3410;
		
	3410:
		FeedCar.AbsMove(Config.pos_StartPoint + 10, 40);
		step := step + 1;
		
	3411:
		IF (FeedCar.bBuzy OR FeedCar.bError) THEN
			step := step + 1;
		END_IF
		
	3412:
		IF FeedCar.bDone  THEN
			step := step + 1;
		ELSIF FeedCar.bError THEN
			step := step + 10000;
		END_IF
		
	3413:
		step := 3420;
		
	3420:
		Hydraulic.CarLift_Down(0);
		step := step + 1;
		
	3421:
		IF (Hydraulic.bBuzy OR Hydraulic.bError) THEN
			step := step + 1;
		END_IF
		
	3422:
		IF Hydraulic.bDone THEN
			step := step + 1;
		ELSIF Hydraulic.bError THEN
			step := step + 10000;
		END_IF
		
	3423:
		step := 3430;
	
	3430:
		pmsg.Push_Error(
				WStrConcat(
					"FeedMain:進料寬度錯誤$n註冊值:",
					TO_WSTRING(Wide_Size),
					"$n測量值:",
					TO_WSTRING(FeedCar.rFindPos),
					"$nAT:",
					TO_WSTRING(step)
				)
			);
		step := step + 10000;

END_CASE
END_ACTION

ACTION Step_8000_Jog_Start:
(*====================================
				Jog模式
  ====================================*) 
//IF ((Hmi.Mode_Select = 1 OR Hmi.Mode_Select = 2)) AND step >= 8000 AND step < 9800 THEN
//	step := 9800;
//END_IF

IF SystemError THEN
	Hmi_Web.Roller_Fwd_S := FALSE;
	Hmi_Web.Roller_Rev_S := FALSE;
	Hmi_Web.Roller_Fwd := FALSE;
	Hmi_Web.Roller_Rev := FALSE;
	
	Hmi_Web.Roller_Up_S := FALSE;
	Hmi_Web.Roller_Down_S := FALSE;
	Hmi_Web.Roller_Up := FALSE;
	Hmi_Web.Roller_Down := FALSE;
	
	Hmi_Web.Car_Fwd_S := FALSE;
	Hmi_Web.Car_Rev_S := FALSE;
	Hmi_Web.Car_Fwd := FALSE;
	Hmi_Web.Car_Rev := FALSE;
	
	Hmi_Web.Car_Up_S := FALSE;
	Hmi_Web.Car_Down_S := FALSE;
	Hmi_Web.Car_Up := FALSE;
	Hmi_Web.Car_Down := FALSE;
	
	Hmi_Web.StopPin_Up_S := FALSE;
	Hmi_Web.StopPin_Down_S := FALSE;
	Hmi_Web.StopPin_Up := FALSE;
	Hmi_Web.StopPin_Down := FALSE;
	
	Hmi_Web.Pull_over_Push_S := FALSE;
	Hmi_Web.Pull_over_Push := FALSE;
END_IF

step_8100_Roller_in();
step_8200_Car();
step_8300_StopPin();
step_8400_PullOver();
step_8500_Roller_Out();

CASE step OF
	8000: // jog按鍵
		bReady := FALSE;
		step := step + 1;
		
	8001:
		CASE Hmi_Web.Site_Select OF
			e_Jog_Site_Select.Input_site:
				IF Hmi_Web.Roller_Fwd THEN
					step := 8100;
				ELSIF Hmi_Web.Roller_Rev THEN
					step := 8120;
				ELSIF Hmi_Web.Roller_Up THEN
					step := 8140;
				ELSIF Hmi_Web.Roller_Down THEN
					step := 8160;
					
				ELSIF Hmi_Web.Car_Fwd THEN
					step := 8200;
				ELSIF Hmi_Web.Car_Rev THEN
					step := 8220;
				ELSIF Hmi_Web.Car_Up THEN
					step := 8240;
				ELSIF Hmi_Web.Car_Down THEN
					step := 8260;
					
				ELSIF Hmi_Web.StopPin_Up THEN
					step := 8300;
				ELSIF Hmi_Web.StopPin_Down THEN
					step := 8320;
					
				ELSIF Hmi_Web.Pull_over_Push THEN
					step := 8400;
				END_IF
				
			e_Jog_Site_Select.Output_Site:
				IF Hmi_Web.Roller_Fwd THEN
					step := 8500;
				ELSIF Hmi_Web.Roller_Rev THEN
					step := 8520;
				ELSIF Hmi_Web.Roller_Up THEN
					step := 8540;
				ELSIF Hmi_Web.Roller_Down THEN
					step := 8560;
				END_IF
				
		END_CASE
		
		IF (Input.Feed_Start) OR SystemError THEN 
			step := 9800;
		END_IF
		
	
	9800:
		Hmi_Web.Roller_Fwd_S := FALSE;
		Hmi_Web.Roller_Rev_S := FALSE;
		Hmi_Web.Roller_Fwd := FALSE;
		Hmi_Web.Roller_Rev := FALSE;
		
		Hmi_Web.Roller_Up_S := FALSE;
		Hmi_Web.Roller_Down_S := FALSE;
		Hmi_Web.Roller_Up := FALSE;
		Hmi_Web.Roller_Down := FALSE;
		
		Hmi_Web.Car_Fwd_S := FALSE;
		Hmi_Web.Car_Rev_S := FALSE;
		Hmi_Web.Car_Fwd := FALSE;
		Hmi_Web.Car_Rev := FALSE;
		
		Hmi_Web.Car_Up_S := FALSE;
		Hmi_Web.Car_Down_S := FALSE;
		Hmi_Web.Car_Up := FALSE;
		Hmi_Web.Car_Down := FALSE;
		
		Hmi_Web.StopPin_Up_S := FALSE;
		Hmi_Web.StopPin_Down_S := FALSE;
		Hmi_Web.StopPin_Up := FALSE;
		Hmi_Web.StopPin_Down := FALSE;
		
		Hmi_Web.Pull_over_Push_S := FALSE;
		Hmi_Web.Pull_over_Push := FALSE;
		
		step := step + 1;
		
	
		
	9801:
// 		pmsg.Push_Info("退出手動模式");
		step := 0;
		
END_CASE
END_ACTION

ACTION step_8100_Roller_in:
(*====================================
		Group A X軸 Jog模式
  ====================================*) 

CASE step OF
(*====================================
				正方向
  ====================================*)
	8100:
		FeedRoller.Jog_Rev();
		step := step + 1;
		
		
	8101:
		IF NOT Hmi_Web.Roller_Fwd THEN
			step := 8109;
		ELSIF FeedRoller.bBuzy OR FeedRoller.bError THEN
			step := step + 1;
		END_IF
		
	8102:
		IF FeedRoller.bError OR NOT Hmi_Web.Roller_Fwd THEN
			step:=8109;
		END_IF
		
	8109:
		FeedRoller.Jog_Stop();
		step:=8001;
		
(*====================================
				負方向
  ====================================*) 
		
	8120:
		FeedRoller.Jog_Fwd();
		step := step + 1;
		
		
	8121:
		IF NOT Hmi_Web.Roller_Rev THEN
			step := 8129;
		ELSIF FeedRoller.bBuzy OR FeedRoller.bError THEN
			step := step + 1;
		END_IF
		
	8122:
		
		IF FeedRoller.bError OR NOT Hmi_Web.Roller_Rev THEN
			step:=8129;
		END_IF
		
	8129:
		FeedRoller.Jog_Stop();
		step:=8001;
		
(*====================================
				上升
  ====================================*)
	8140:
		FeedRoller.Jog_Up();
		step := step + 1;
		
		
	8141:
		IF FeedRoller.bBuzy OR FeedRoller.bError THEN
			step := step + 1;
		END_IF
		
	8142:
		IF FeedRoller.bDone OR FeedRoller.bError THEN
			step:=8149;
		END_IF
		
	8149:
		step:=8001;
		
(*====================================
				下降
  ====================================*) 
		
	8160:
		FeedRoller.Jog_Down();
		step := step + 1;
		
		
	8161:
		IF FeedRoller.bBuzy OR FeedRoller.bError THEN
			step := step + 1;
		END_IF
		
	8162:
		IF FeedRoller.bDone OR FeedRoller.bError THEN
			step:=8169;
		END_IF
		
	8169:
		step:=8001;

END_CASE

Hmi_Web.Roller_Fwd_S	:= step >= 8100 AND step < 8109;
Hmi_Web.Roller_Rev_S	:= step >= 8120 AND step < 8129;
Hmi_Web.Roller_Up_S		:= step >= 8140 AND step < 8149;
Hmi_Web.Roller_Down_S	:= step >= 8160 AND step < 8169;
END_ACTION

ACTION step_8200_Car:
(*====================================
		Group A X軸 Jog模式
  ====================================*) 

CASE step OF
(*====================================
				正方向
  ====================================*)
	8200:
		IF FeedCar.bHome THEN
			FeedCar.AbsMove(config.pos_Workpiace_FeedPoint,  Hmi_Web.Speed_Select);
			step := step + 1;
		ELSE
			step := 8209;
		END_IF
		
		
	8201:
		IF NOT Hmi_Web.Car_Fwd THEN
			step := 8209;
		ELSIF FeedCar.bBuzy OR FeedCar.bError THEN
			step := step + 1;
		END_IF
		
	8202:
		IF FeedCar.bDone OR FeedCar.bError OR NOT Hmi_Web.Car_Fwd THEN
			step:=8209;
		END_IF
		
	8209:
		FeedCar.Stop();
		IF NOT Hmi_Web.Car_Fwd THEN
			step:=8001;
		END_IF
		
(*====================================
				負方向
  ====================================*) 
		
	8220:
		IF FeedCar.bHome THEN
			FeedCar.AbsMove(0,  Hmi_Web.Speed_Select);
		ELSE
			FeedCar.Homing();
		END_IF
		step := step + 1;
		
		
	8221:
		IF NOT Hmi_Web.Car_Rev THEN
			step := 8229;
		ELSIF FeedCar.bBuzy OR FeedCar.bError THEN
			step := step + 1;
		END_IF
		
	8222:
		IF FeedCar.bDone OR FeedCar.bError OR NOT Hmi_Web.Car_Rev THEN
			step:=8229;
		END_IF
		
	8229:
		FeedCar.Stop();
		IF NOT Hmi_Web.Car_Rev THEN
			step:=8001;
		END_IF
		
(*====================================
				上升
  ====================================*) 
	8240:
		Hydraulic.CarLift_Up(TO_WORD(Hmi_Web.Module_Select));
		step := step + 1;
		
		
	8241:
		IF NOT Hmi_Web.Car_Up THEN
			step := 8249;
		ELSIF Hydraulic.bBuzy OR Hydraulic.bError THEN
			step := step + 1;
		END_IF
		
	8242:
		IF Hydraulic.bDone OR Hydraulic.bError OR NOT Hmi_Web.Car_Up THEN
			step:=8249;
		END_IF
		
	8249:
		Hydraulic.Stop();
		IF NOT Hmi_Web.Car_Up THEN
			step:=8001;
		END_IF
		
(*====================================
				下降
  ====================================*) 
	8260:
		Hydraulic.CarLift_Down(TO_WORD(Hmi_Web.Module_Select));
		step := step + 1;
		
		
	8261:
		IF NOT Hmi_Web.Car_Down THEN
			step := 8269;
		ELSIF Hydraulic.bBuzy OR Hydraulic.bError THEN
			step := step + 1;
		END_IF
		
	8262:
		IF Hydraulic.bDone OR Hydraulic.bError OR NOT Hmi_Web.Car_Down THEN
			step:=8269;
		END_IF
		
	8269:
		Hydraulic.Stop();
		IF NOT Hmi_Web.Car_Down THEN
			step:=8001;
		END_IF

END_CASE

Hmi_Web.Car_Fwd_S	:= step >= 8200 AND step < 8209;
Hmi_Web.Car_Rev_S	:= step >= 8220 AND step < 8229;
Hmi_Web.Car_Up_S	:= step >= 8240 AND step < 8249;
Hmi_Web.Car_Down_S	:= step >= 8260 AND step < 8269;
END_ACTION

ACTION step_8300_StopPin:
(*====================================
		Group A X軸 Jog模式
  ====================================*) 

CASE step OF
(*====================================
				PIN上
  ====================================*)
	8300:
		StopPin.Up(TO_WORD(Hmi_Web.Module_Select));
		step := step + 1;
		
		
	8301:
		IF StopPin.bDone OR StopPin.bError OR NOT Hmi_Web.StopPin_Up THEN
			step:=8309;
		END_IF
	
	8309:
		IF NOT Hmi_Web.StopPin_Up THEN
			step:=8001;
		END_IF
		
		
(*====================================
				PIN下
  ====================================*)
		
	8320:
		StopPin.Down(TO_WORD(Hmi_Web.Module_Select));
		step := step + 1;
		
		
	8321:
		IF StopPin.bDone OR StopPin.bError OR NOT Hmi_Web.StopPin_Down THEN
			step:=8329;
		END_IF
	
	8329:
		IF NOT Hmi_Web.StopPin_Down THEN
			step:=8001;
		END_IF
		
END_CASE


Hmi_Web.StopPin_Up_S	:= step >= 8300 AND step < 8309;
Hmi_Web.StopPin_Down_S	:= step >= 8320 AND step < 8329;
END_ACTION

ACTION step_8400_PullOver:
(*====================================
		Group A X軸 Jog模式
  ====================================*) 

CASE step OF
(*====================================
				正方向
  ====================================*)
	8400:
		Hydraulic.Over_Pull_Jog();
		step := step + 1;
		
		
	8401:
		IF Hydraulic.bDone1 OR NOT Hmi_Web.Pull_over_Push THEN
			step:=8409;
		END_IF
	
	8409:
		IF NOT Hmi_Web.Pull_over_Push THEN
			step:=8001;
		END_IF
		
END_CASE

Hmi_Web.Pull_over_Push_S	:= step >= 8400 AND step < 8409;
END_ACTION

ACTION step_8500_Roller_Out:
(*====================================
		Group A X軸 Jog模式
  ====================================*) 

CASE step OF
(*====================================
				正方向
  ====================================*)
	8500:
		ProductRoller.Jog_Rev();
		step := step + 1;
		
		
	8501:
		IF NOT Hmi_Web.Roller_Fwd THEN
			step := 8509;
		ELSIF ProductRoller.bBuzy OR ProductRoller.bError THEN
			step := step + 1;
		END_IF
		
	8502:
		IF ProductRoller.bError OR NOT Hmi_Web.Roller_Fwd THEN
			step:=8509;
		END_IF
		
	8509:
		ProductRoller.Jog_Stop();
		step:=8001;
		
(*====================================
				負方向
  ====================================*) 
		
 	8520:
		ProductRoller.Jog_Fwd();
		step := step + 1;
		
		
 	8521:
		IF NOT Hmi_Web.Roller_Rev THEN
			step := 8129;
		ELSIF ProductRoller.bBuzy OR ProductRoller.bError THEN
			step := step + 1;
		END_IF
		
 	8522:
		
		IF ProductRoller.bError OR NOT Hmi_Web.Roller_Rev THEN
			step:=8529;
		END_IF
		
 	8529:
		ProductRoller.Jog_Stop();
		step:=8001;
		
(*====================================
				上升
  ====================================*)
 	8540:
		ProductRoller.Jog_Up();
		step := step + 1;
		
		
 	8541:
		IF ProductRoller.bBuzy OR ProductRoller.bError THEN
			step := step + 1;
		END_IF
		
 	8542:
		IF ProductRoller.bDone OR ProductRoller.bError THEN
			step:=8549;
		END_IF
		
 	8549:
		step:=8001;
		
(*====================================
				下降
  ====================================*) 
		
 	8560:
		ProductRoller.Jog_Down();
		step := step + 1;
		
		
 	8561:
		IF ProductRoller.bBuzy OR ProductRoller.bError THEN
			step := step + 1;
		END_IF
		
 	8562:
		IF ProductRoller.bDone OR ProductRoller.bError THEN
			step:=8569;
		END_IF
		
 	8569:
		step:=8001;

END_CASE

Hmi_Web.Roller_Fwd_S	:= step >= 8100 AND step < 8109;
Hmi_Web.Roller_Rev_S	:= step >= 8120 AND step < 8129;
Hmi_Web.Roller_Up_S		:= step >= 8140 AND step < 8149;
Hmi_Web.Roller_Down_S	:= step >= 8160 AND step < 8169;
END_ACTION

ACTION Timer:
tmr01();
END_ACTION

END_PROGRAM

// ---- POUs/功能塊/字串處理功能塊/字串記憶/WStrMem.TcPOU
FUNCTION_BLOCK WStrMem
VAR_INPUT
END_VAR
VAR_OUTPUT
END_VAR
VAR
	mem : WSTRING;
END_VAR

METHOD APPEND : BOOL
VAR_INPUT
	STR : WSTRING;
END_VAR
mem := WCONCAT(mem , STR);
END_METHOD

METHOD INSERT : BOOL
VAR_INPUT
	STR : WSTRING;
END_VAR
mem := WCONCAT(STR, mem);
END_METHOD

PROPERTY READ : WSTRING
GET
READ := mem;
END_GET
END_PROPERTY

METHOD WRITE : BOOL
VAR_INPUT
	STR :WSTRING;
END_VAR
mem := STR;
END_METHOD

END_FUNCTION_BLOCK

// ---- POUs/功能塊/資料庫 Postgre相關/記錄用/程式紀錄/Step_Log.TcPOU
FUNCTION_BLOCK Step_Log
VAR_INPUT
	name : STRING(80);
	step : DINT;
END_VAR
VAR_OUTPUT
END_VAR
VAR
	exec_number : UDINT;
	
	exec_done_number : UDINT;
	
	array_select_number : INT;
	
	_logData_array : ARRAY [0..31] OF StepLog_Struct;

	old_step : DINT;
	
	_logData : StepLog_Struct;

	db_fb_PLCDBCmdEvt : FB_PLCDBCmdEvt(sNetID:= '', tTimeout:= T#5S );
	
	_stPara		: ARRAY [0..3] OF ST_ExpParameter;
	
	_SqlCommand : STRING(1024);
	
	_extrasstr : STRING(255);
	
	_fbJson      : FB_JsonSaxWriter;
END_VAR

IF step <> old_step THEN
	old_step := step;
	
	array_select_number := TO_INT(exec_number MOD 32);
	
	IF array_select_number >= 0 AND array_select_number < 32 THEN
		_logData_array[array_select_number].program_name := name;
		
		_logData_array[array_select_number].step_number := step;
		
		_logData_array[array_select_number].created_at := TO_LINT(F_GetSystemTime());
		
		_logData_array[array_select_number].extras_Srt := _extrasstr;
		
		_extrasstr := '{}';
	END_IF
	
	exec_number := exec_number + 1;
END_IF

IF exec_number > exec_done_number  THEN
	array_select_number := TO_INT(exec_done_number MOD 32);

	IF array_select_number >= 0 AND array_select_number < 32 THEN
			_logData := _logData_array[array_select_number];
			
			// SQL命令
			_SqlCommand := 
		
			'INSERT 
				INTO exp1_program_running_log 
					(program_name, step_number, created_at, detail_data)
				VALUES
					({program_name}, {step_number}, to_timestamp(({created_at} - 116444736000000000) / 10000000.0), {detail_data}::jsonb);
			';
		
		// 設定對應參數
			_stPara[0].sParaName := 'step_number'; 			_stPara[0].eParaType := E_ExpParameterType.Int32; 		_stPara[0].nParaSize := SIZEOF(_logData.step_number);
			_stPara[1].sParaName := 'created_at';			_stPara[1].eParaType := E_ExpParameterType.Int64;		_stPara[1].nParaSize := SIZEOF(_logData.created_at);
			_stPara[2].sParaName := 'program_name'; 		_stPara[2].eParaType := E_ExpParameterType.STRING_; 	_stPara[2].nParaSize := 81;
			_stPara[3].sParaName := 'detail_data'; 			_stPara[3].eParaType := E_ExpParameterType.STRING_; 	_stPara[3].nParaSize := 256;
			
		IF db_fb_PLCDBCmdEvt.Execute(
				hDBID := 3,
				pExpression := ADR(_SqlCommand),			// SQL 命令 ex. SELECT * FROM PlcTest.newtable WHERE ID = {ID}  
				cbExpression := SIZEOF(_SqlCommand),		// SQL 命令字串的長度
				pData:= ADR(_logData),		// 帶入的參數值
				cbData:= SIZEOF(_logData),//itmp, 	// 帶入的參數值大小
				pParameter:= ADR(_stPara), 				// 帶入的參數類型設定  ex.上面命令內的 {ID} 類型設定
				cbParameter:= SIZEOF(_stPara),			// 帶入的參數類型設定的大小
			)  
		THEN
			
			exec_done_number := exec_done_number + 1;
		END_IF
	END_IF
END_IF

{attribute 'suppress_wrn_C0410'}
PROPERTY fbJson : REFERENCE TO FB_JsonSaxWriter
GET
fbJson REF= _fbJson;
END_GET
END_PROPERTY

METHOD JsonOutput : BOOL
VAR_INPUT
END_VAR
fbJson.EndObject();
_extrasstr := fbJson.GetDocument();
fbJson.ResetDocument();
END_METHOD

END_FUNCTION_BLOCK

// ---- POUs/功能塊/資料庫 Postgre相關/動作資料/ReadSQLData.TcPOU
PROGRAM ReadSQLData
VAR
	step : INT;	

	_fb_PLCDBCmdEvt : FB_PLCDBCmdEvt(sNetID:= '', tTimeout:= T#5S );

	
	_SqlCommand : STRING(1024);
	
	// 讀回的資料筆數
	read_num: UDINT;
	
	// 帶入參數
	_stPara		: ARRAY [0..5] OF ST_ExpParameter;
	
	tcMessage     : I_TcMessage;
	
	database_server_id: UDINT := 2;
	
	_uuid : STRING(36);
	
	_DataExists :BOOL;
	
	_tmp_db_Steel_Status : sc_db_Steel_Status;
	
	_waitLoading_Pos : sc_db_Set_Work_Order_WaitLoading_Pos;
	
	test: PVOID;
	TmrWdt: TON;
	_tmp_number: INT;
END_VAR

VAR_OUTPUT
	bBuzy	: BOOL;
	bDone	: BOOL;
	bError	: BOOL;
	
	fNext_XPos	: LREAL;
END_VAR


bBuzy := step > 0 AND step < 10000;

bError := step > 10000;

IF bBuzy OR bError  THEN
	bDone := FALSE;
END_IF

TmrWdt(in := bBuzy, PT:=T#20S);
IF TmrWdt.Q THEN
	pMsg.Push_alarm(
				ErrorCodeConver.Str2("ReadSQLData", ":功能執行超時", TO_DWORD(step))
			);
	step := step + 10000;
END_IF

IF step = 0 THEN
	RETURN;
END_IF



Stap_0100_Get_Work_Order();
Stap_1000_Set_Work_Order_Status();
Stap_1100_Set_Work_Order_WaitLoading_Pos();

METHOD Get_WorkkOrder
VAR_INPUT
	Status : STRING := 'holding';
END_VAR
bdone := FALSE;

_uuid := Status;

step := 100;
END_METHOD

METHOD Set_Work_Order_2_inSide
VAR_INPUT
	id : UINT;
	
	(*
	finish 加工完成
	inSide 入料  
	holding 暫存中(在吊掛區等待進入料架)
	machining 加工中
	alignment 無靠邊插單
	inserts 插單
	waitLoading 等待上料(在料架上等待，後進入機台)
	waitUnloading 等待下料(在料架上等待，後進入出料吊掛區或其他機台)
	paired 已配對
	pairing 配對中
	pairedFailed 配對失敗
	dxfTransferring DXF 傳輸中
	connectedFailed 連線失敗
	transformFailed 轉換失敗
	waitPaired 等待配對
	pairedCancel 配對取消
	unknown 未知
	*)
// 	status : STRING(80) := '';
	
	(*
		holdingEntranceRack 吊掛入料區
		entranceRack 機器入料區
		holdingExitRack 吊掛出料區
		exitRack 機器出料區
		machine 機台內
	*)
// 	location : STRING(80) := '';
END_VAR
_tmp_db_Steel_Status.uuid := ProjectData.WorkOrder_At_waitLoading[id].steel_id;

_tmp_db_Steel_Status.steel_status := 'inSide';

_tmp_db_Steel_Status.steel_location := 'entranceRack';

step := 1000;
END_METHOD

METHOD Set_Work_Order_2_waitLoading
VAR_INPUT
	id : UINT;
	
	(*
	finish 加工完成
	inSide 入料  
	holding 暫存中(在吊掛區等待進入料架)
	machining 加工中
	alignment 無靠邊插單
	inserts 插單
	waitLoading 等待上料(在料架上等待，後進入機台)
	waitUnloading 等待下料(在料架上等待，後進入出料吊掛區或其他機台)
	paired 已配對
	pairing 配對中
	pairedFailed 配對失敗
	dxfTransferring DXF 傳輸中
	connectedFailed 連線失敗
	transformFailed 轉換失敗
	waitPaired 等待配對
	pairedCancel 配對取消
	unknown 未知
	*)
// 	status : STRING(80) := '';
	
	(*
		holdingEntranceRack 吊掛入料區
		entranceRack 入料區
		holdingExitRack 吊掛出料區
		exitRack 出料區
		machine 機台內
	*)
// 	location : STRING(80) := '';
END_VAR
_tmp_db_Steel_Status.uuid := ProjectData.WorkOrder_At_holding[id].steel_id;

_tmp_db_Steel_Status.steel_status := 'waitLoading';

_tmp_db_Steel_Status.steel_location := '';

step := 1000;
END_METHOD

METHOD Set_Work_Order_Status
VAR_INPUT
	uuid : STRING(36);
	
	status		: STRING;
	
	location	: STRING;
	(*
	finish 加工完成
	inSide 入料  
	holding 暫存中(在吊掛區等待進入料架)
	machining 加工中
	alignment 無靠邊插單
	inserts 插單
	waitLoading 等待上料(在料架上等待，後進入機台)
	waitUnloading 等待下料(在料架上等待，後進入出料吊掛區或其他機台)
	paired 已配對
	pairing 配對中
	pairedFailed 配對失敗
	dxfTransferring DXF 傳輸中
	connectedFailed 連線失敗
	transformFailed 轉換失敗
	waitPaired 等待配對
	pairedCancel 配對取消
	unknown 未知
	*)
// 	status : STRING(80) := '';
	
	(*
		holdingEntranceRack 吊掛入料區
		entranceRack 入料區
		holdingExitRack 吊掛出料區
		exitRack 出料區
		machine 機台內
	*)
// 	location : STRING(80) := '';
END_VAR
_tmp_db_Steel_Status.uuid := uuid;

_tmp_db_Steel_Status.steel_status := status;

_tmp_db_Steel_Status.steel_location := location;

step := 1000;
END_METHOD

METHOD  Set_Work_Order_WaitLoading_Pos : BOOL
VAR_INPUT
	id : uint;
	Pos : LREAL;
END_VAR
_waitLoading_Pos.uuid := ProjectData.WorkOrder_At_holding[id].steel_id;
_waitLoading_Pos.Pos := Pos;

step := 1100;
END_METHOD

ACTION Stap_0100_Get_Work_Order:
CASE step OF
	100:
		step := step + 1;

	101:
		// SQL命令
		_SqlCommand := 
		'
		SELECT 
			"sequence_number",
			s.height,
			s.width,
			CAST("part_nest_id" as char(36)),
			waitloading_at_pos
		FROM
			"public"."work_order_data" 
		LEFT JOIN 
			"public"."steeldata" s 
		ON 
			s.id = part_nest_id::uuid
		WHERE
 			"steel_status" = $'holding$' AND work_order_data.processing_project_id = {id}
		ORDER BY 
			"sequence_number"
		';
	
		// 設定對應參數
 		_stPara[0].sParaName := 'id'; 			_stPara[0].eParaType := E_ExpParameterType.STRING_; 		_stPara[0].nParaSize := SIZEOF(_uuid);
		step := step + 1;
		
	102:
		IF 
			_fb_PLCDBCmdEvt.ExecuteDataReturn(
				hDBID := database_server_id,
				pExpression := ADR(_SqlCommand),			// SQL 命令 ex. SELECT * FROM PlcTest.newtable WHERE ID = {ID}  
				cbExpression := SIZEOF(_SqlCommand),		// SQL 命令字串的長度
				pData:= ADR(Input.Feed_WorkOrder_UUID),							// 帶入的參數值
				cbData:= SIZEOF(Input.Feed_WorkOrder_UUID),						// 帶入的參數值大小
				pParameter:= ADR(_stPara), 					// 帶入的參數類型設定  ex.上面命令內的 {ID} 類型設定
				cbParameter:= SIZEOF(_stPara[0]) * 1,		// 帶入的參數類型設定的大小
				nStartIndex := 0,
				nRecordCount := 32,
				pReturnData := ADR(ProjectData.WorkOrder_At_holding),
				cbReturnData := SIZEOF(ProjectData.WorkOrder_At_holding),
				pRecords := ADR(read_num)
			) 
		THEN
			IF _fb_PLCDBCmdEvt.bError THEN
				tcMessage := _fb_PLCDBCmdEvt.ipTcResult;
				step := step + 10000;
			ELSE
				ProjectData.WorkOrder_Nunber_At_holding := TO_UINT(read_num);
				step := step + 1;
			END_IF
			
		END_IF
		
	103:
		step := 110;
		
	110:
		step := 111;
		
	111:
		// SQL命令
		_SqlCommand := 
		'
		SELECT 
			"sequence_number",
			s.height,
			s.width,
			CAST("part_nest_id" as char(36)),
			waitloading_at_pos
		FROM
			"public"."work_order_data" 
		LEFT JOIN 
			"public"."steeldata" s 
		ON 
			s.id = part_nest_id::UUID
		WHERE
 			"steel_status" = $'waitLoading$'
		ORDER BY 
			"sequence_number"
		';
	
		step := step + 1;
		
	112:
		IF 
			_fb_PLCDBCmdEvt.ExecuteDataReturn(
				hDBID := database_server_id,
				pExpression := ADR(_SqlCommand),			// SQL 命令 ex. SELECT * FROM PlcTest.newtable WHERE ID = {ID}  
				cbExpression := SIZEOF(_SqlCommand),		// SQL 命令字串的長度
				pData:= 0,									// 帶入的參數值
				cbData:= 0,									// 帶入的參數值大小
				pParameter:= 0,					// 帶入的參數類型設定  ex.上面命令內的 {ID} 類型設定
				cbParameter:= 0,		// 帶入的參數類型設定的大小
// 				pData:= ADR(_uuid),							// 帶入的參數值
// 				cbData:= SIZEOF(_uuid),						// 帶入的參數值大小
// 				pParameter:= ADR(_stPara), 					// 帶入的參數類型設定  ex.上面命令內的 {ID} 類型設定
// 				cbParameter:= SIZEOF(_stPara[0]) * 1,		// 帶入的參數類型設定的大小
				nStartIndex := 0,
				nRecordCount := 32,
				pReturnData := ADR(ProjectData.WorkOrder_At_waitLoading),
				cbReturnData := SIZEOF(ProjectData.WorkOrder_At_waitLoading),
				pRecords := ADR(read_num)
			) 
		THEN
			IF _fb_PLCDBCmdEvt.bError THEN
				tcMessage := _fb_PLCDBCmdEvt.ipTcResult;
				step := step + 10000;
			ELSE
				ProjectData.WorkOrder_Nunber_At_waitLoading := TO_UINT(read_num);
				step := step + 1;
			END_IF
			
		END_IF
		
	113:
		step := 120;
		
	120:
		step := 121;
		
	121:
		// SQL命令
		_SqlCommand := 
		'
		SELECT 
			Count(*)::int2
		FROM
			public.work_order_data
		WHERE
 			steel_status = $'machine$'
		';
	
		step := step + 1;
		
	122:
		IF 
			_fb_PLCDBCmdEvt.ExecuteDataReturn(
				hDBID := database_server_id,
				pExpression := ADR(_SqlCommand),			// SQL 命令 ex. SELECT * FROM PlcTest.newtable WHERE ID = {ID}  
				cbExpression := SIZEOF(_SqlCommand),		// SQL 命令字串的長度
				pData:= 0,									// 帶入的參數值
				cbData:= 0,									// 帶入的參數值大小
				pParameter:= 0,					// 帶入的參數類型設定  ex.上面命令內的 {ID} 類型設定
				cbParameter:= 0,		// 帶入的參數類型設定的大小
// 				pData:= ADR(_uuid),							// 帶入的參數值
// 				cbData:= SIZEOF(_uuid),						// 帶入的參數值大小
// 				pParameter:= ADR(_stPara), 					// 帶入的參數類型設定  ex.上面命令內的 {ID} 類型設定
// 				cbParameter:= SIZEOF(_stPara[0]) * 1,		// 帶入的參數類型設定的大小
				nStartIndex := 0,
				nRecordCount := 1,
				pReturnData := ADR(ProjectData.WorkOrder_Nunber_At_Machining),
				cbReturnData := SIZEOF(ProjectData.WorkOrder_Nunber_At_Machining),
				pRecords := ADR(read_num)
			) 
		THEN
			IF _fb_PLCDBCmdEvt.bError THEN
				tcMessage := _fb_PLCDBCmdEvt.ipTcResult;
				step := step + 10000;
			ELSE
				step := step + 1;
			END_IF
			
		END_IF
		
	123:
		step := 130;
		
	130:
		bDone := TRUE;
		step := 0;
END_CASE
END_ACTION

ACTION Stap_1000_Set_Work_Order_Status:
CASE step OF
	1000:
		IF len(_tmp_db_Steel_Status.steel_location) > 0 OR len(_tmp_db_Steel_Status.steel_status) > 0 THEN
			step := step + 1;
		ELSE
			step := step + 10000;
		END_IF
		
	1001:
		step := 1010;

	1010:
		_SqlCommand := ' UPDATE work_order_data SET ';
		IF len(_tmp_db_Steel_Status.steel_status) > 0 THEN
			_SqlCommand := CONCAT(STR1:= _SqlCommand, STR2:= 'steel_status = {status}');
		END_IF
		IF len(_tmp_db_Steel_Status.steel_location) > 0 THEN
			_SqlCommand := CONCAT(STR1:= _SqlCommand, STR2:= ', steel_location = {location}');
		END_IF
		// SQL命令
		_SqlCommand := CONCAT(STR1:= _SqlCommand, STR2:= ' WHERE part_nest_id = {id}');
	
		// 設定對應參數
 		_stPara[0].sParaName := 'id'; 			_stPara[0].eParaType := E_ExpParameterType.STRING_; 		_stPara[0].nParaSize := 37;
		_stPara[1].sParaName := 'status'; 		_stPara[1].eParaType := E_ExpParameterType.STRING_; 		_stPara[1].nParaSize := 81;
		_stPara[2].sParaName := 'location'; 	_stPara[2].eParaType := E_ExpParameterType.STRING_; 		_stPara[2].nParaSize := 81;
		step := step + 1;
		
	1011:
		IF 
			_fb_PLCDBCmdEvt.Execute(
				hDBID := database_server_id,
				pExpression := ADR(_SqlCommand),			// SQL 命令 ex. SELECT * FROM PlcTest.newtable WHERE ID = {ID}  
				cbExpression := SIZEOF(_SqlCommand),		// SQL 命令字串的長度
				pData:= ADR(_tmp_db_Steel_Status),			// 帶入的參數值
				cbData:= SIZEOF(_tmp_db_Steel_Status),		// 帶入的參數值大小
				pParameter:= ADR(_stPara), 					// 帶入的參數類型設定  ex.上面命令內的 {ID} 類型設定
				cbParameter:= SIZEOF(_stPara[0]) * 3,		// 帶入的參數類型設定的大小
			) 
		THEN
			IF _fb_PLCDBCmdEvt.bError THEN
				tcMessage := MsgMain._fb_PLCDBCmdEvt.ipTcResult;
				step := step + 10000;
			ELSE
				step := step + 1;
			END_IF
		END_IF
		
	1012:
		pMsg.Push_Info(WStrConcat(
				"Set_Steel_Start: ",
				WLEFT(STR:= TO_WSTRING(_uuid), SIZE:= 8),
				" :狀態設定為:",
				TO_WSTRING(_tmp_db_Steel_Status.steel_status)
				));
		bDone :=TRUE;
		step := 0;
END_CASE
END_ACTION

ACTION Stap_1100_Set_Work_Order_WaitLoading_Pos:
CASE step OF
	1100:
		step := 1110;

	1110:
		_SqlCommand := ' 
			UPDATE work_order_data 
			SET waitloading_at_pos = {pos}
			WHERE part_nest_id = {id}
			';
			
		// 設定對應參數
 		_stPara[0].sParaName := 'id'; 			_stPara[0].eParaType := E_ExpParameterType.STRING_; 		_stPara[0].nParaSize := 37;
		_stPara[1].sParaName := 'pos'; 			_stPara[1].eParaType := E_ExpParameterType.Double64; 		_stPara[1].nParaSize := 8;
		step := step + 1;
		
	1111:
		IF 
			MsgMain._fb_PLCDBCmdEvt.Execute(
				hDBID := database_server_id,
				pExpression := ADR(_SqlCommand),			// SQL 命令 ex. SELECT * FROM PlcTest.newtable WHERE ID = {ID}  
				cbExpression := SIZEOF(_SqlCommand),		// SQL 命令字串的長度
				pData:= ADR(_waitLoading_Pos),			// 帶入的參數值
				cbData:= SIZEOF(_waitLoading_Pos),		// 帶入的參數值大小
				pParameter:= ADR(_stPara), 					// 帶入的參數類型設定  ex.上面命令內的 {ID} 類型設定
				cbParameter:= SIZEOF(_stPara[0]) * 2,		// 帶入的參數類型設定的大小
			) 
		THEN
			IF MsgMain._fb_PLCDBCmdEvt.bError THEN
				tcMessage := MsgMain._fb_PLCDBCmdEvt.ipTcResult;
				step := step + 10000;
			ELSE
				step := step + 1;
			END_IF
		END_IF
		
	1112:
		bDone :=TRUE;
		step := 0;
END_CASE
END_ACTION

END_PROGRAM

// ---- POUs/功能塊/ErrorCodeConver.TcPOU
PROGRAM ErrorCodeConver
VAR
	
END_VAR

METHOD StoberErrorCode : WSTRING
VAR_INPUT
	Name : WSTRING;
	Event : UDINT;
	Cause : UDINT;
END_VAR

VAR
	strtmp1: WSTRING;
	strtmp2: WSTRING;
END_VAR




strtmp2 := WCONCAT(STR1:= Name, STR2:= ":錯誤 Event:");

strtmp1 := UDINT_TO_WSTRING(Event);

strtmp2 := WCONCAT(STR1:= strtmp2, STR2:= strtmp1 );

strtmp2:= WCONCAT(STR1:= strtmp2, STR2:= "Cause:");

strtmp1 := UDINT_TO_WSTRING(Cause);

strtmp2:= WCONCAT(STR1:= strtmp2, STR2:= strtmp1);

// 輸出結果字串

StoberErrorCode := strtmp2;
END_METHOD

METHOD Str1 : WSTRING
VAR_INPUT
	str0 : WSTRING;
	ErrorCode :DWORD;
END_VAR

VAR
	strtmp1: STRING;
	strtmp2: WSTRING;
END_VAR
IF ErrorCode > 16#FFFF THEN
	strtmp1 := DWORD_TO_HEXSTR(in:= ErrorCode, iPrecision:= 8, bLoCase:= FALSE);
ELSE
	strtmp1 := DWORD_TO_HEXSTR(in:= ErrorCode, iPrecision:= 4, bLoCase:= FALSE);
END_IF

strtmp2 := STRING_TO_WSTRING(strtmp1);

strtmp2 := WCONCAT(STR1:= "(", STR2:= strtmp2);

strtmp2 := WCONCAT(STR1:= strtmp2, STR2:= ")" );

Str1:= WCONCAT(STR1:= str0, STR2:= strtmp2);
END_METHOD

METHOD Str2 : WSTRING
VAR_INPUT
	str0 : WSTRING := "";
	str1 : WSTRING := "";
	ErrorCode :DWORD;
END_VAR

VAR
	strtmp1: STRING;
	strtmp2: WSTRING;
END_VAR
IF ErrorCode > 16#FFFF THEN
	strtmp1 := DWORD_TO_HEXSTR(in:= ErrorCode, iPrecision:= 8, bLoCase:= FALSE);
ELSE
	strtmp1 := DWORD_TO_HEXSTR(in:= ErrorCode, iPrecision:= 4, bLoCase:= FALSE);
END_IF

strtmp2 := STRING_TO_WSTRING(strtmp1);

strtmp2 := WCONCAT(STR1:= "(", STR2:= strtmp2);

strtmp2 := WCONCAT(STR1:= strtmp2, STR2:= ")" );

strtmp2:= WCONCAT(STR1:= str1, STR2:= strtmp2);

Str2:= WCONCAT(STR1:= str0, STR2:= strtmp2);
END_METHOD

METHOD Str3 : WSTRING
VAR_INPUT
	str0 : WSTRING := "";
	str1 : WSTRING := "";
	str2 : WSTRING := "";
	ErrorCode :DWORD;
END_VAR

VAR
	strtmp1: STRING;
	strtmp2: WSTRING;
END_VAR
IF ErrorCode > 16#FFFF THEN
	strtmp1 := DWORD_TO_HEXSTR(in:= ErrorCode, iPrecision:= 8, bLoCase:= FALSE);
ELSE
	strtmp1 := DWORD_TO_HEXSTR(in:= ErrorCode, iPrecision:= 4, bLoCase:= FALSE);
END_IF

strtmp2 := STRING_TO_WSTRING(strtmp1);

strtmp2 := WCONCAT(STR1:= "(", STR2:= strtmp2);

strtmp2 := WCONCAT(STR1:= strtmp2, STR2:= ")" );

strtmp2:= WCONCAT(STR1:= str2, STR2:= strtmp2);

strtmp2:= WCONCAT(STR1:= str1, STR2:= strtmp2);

Str3:= WCONCAT(STR1:= str0, STR2:= strtmp2);
END_METHOD

METHOD Str4 : WSTRING
VAR_INPUT
	str0 : WSTRING := "";
	str1 : WSTRING := "";
	str2 : WSTRING := "";
	str3 : WSTRING := "";
	ErrorCode :DWORD;
END_VAR

VAR
	strtmp1: STRING;
	strtmp2: WSTRING;
END_VAR
IF ErrorCode > 16#FFFF THEN
	strtmp1 := DWORD_TO_HEXSTR(in:= ErrorCode, iPrecision:= 8, bLoCase:= FALSE);
ELSE
	strtmp1 := DWORD_TO_HEXSTR(in:= ErrorCode, iPrecision:= 4, bLoCase:= FALSE);
END_IF

strtmp2 := STRING_TO_WSTRING(strtmp1);

strtmp2 := WCONCAT(STR1:= "(", STR2:= strtmp2);

strtmp2 := WCONCAT(STR1:= strtmp2, STR2:= ")" );

strtmp2:= WCONCAT(STR1:= str3, STR2:= strtmp2);

strtmp2:= WCONCAT(STR1:= str2, STR2:= strtmp2);

strtmp2:= WCONCAT(STR1:= str1, STR2:= strtmp2);

Str4:= WCONCAT(STR1:= str0, STR2:= strtmp2);
END_METHOD

METHOD Str5 : WSTRING
VAR_INPUT
	str0 : WSTRING := "";
	str1 : WSTRING := "";
	str2 : WSTRING := "";
	str3 : WSTRING := "";
	str4 : WSTRING := "";
	ErrorCode :DWORD;
END_VAR

VAR
	strtmp1: STRING;
	strtmp2: WSTRING;
END_VAR
IF ErrorCode > 16#FFFF THEN
	strtmp1 := DWORD_TO_HEXSTR(in:= ErrorCode, iPrecision:= 8, bLoCase:= FALSE);
ELSE
	strtmp1 := DWORD_TO_HEXSTR(in:= ErrorCode, iPrecision:= 4, bLoCase:= FALSE);
END_IF

strtmp2 := STRING_TO_WSTRING(strtmp1);

strtmp2 := WCONCAT(STR1:= "(", STR2:= strtmp2);

strtmp2 := WCONCAT(STR1:= strtmp2, STR2:= ")" );

strtmp2:= WCONCAT(STR1:= str4, STR2:= strtmp2);

strtmp2:= WCONCAT(STR1:= str3, STR2:= strtmp2);

strtmp2:= WCONCAT(STR1:= str2, STR2:= strtmp2);

strtmp2:= WCONCAT(STR1:= str1, STR2:= strtmp2);

Str5:= WCONCAT(STR1:= str0, STR2:= strtmp2);
END_METHOD

END_PROGRAM

// ---- MSG/通知訊息/MsgMain.TcPOU
PROGRAM MsgMain
VAR
	MsgNum			: USINT;
	
	_fb_PLCDBCmdEvt : FB_PLCDBCmdEvt(sNetID:= '', tTimeout:= T#5S );
	
	msg		: MsgStruct;
	
	_SqlCommand : STRING(255);
	
	_stPara		: ARRAY [0..5] OF ST_ExpParameter;
	
	tcMessage     : I_TcMessage;
	
	itmp: UINT;
	
	msgtmp		: MsgStruct_RAW;
	
	str : POINTER TO ARRAY[0..159] OF BYTE;
	
	str2 : POINTER TO ARRAY[0..159] OF BYTE;
	
	str3 : POINTER TO ARRAY[0..499] OF BYTE;
END_VAR

IF msgbuff.DoneNumber < msgbuff.evenNumber THEN
	MsgNum := ULINT_TO_USINT(msgbuff.DoneNumber MOD 16);

	msg := msgbuff.messageList[MsgNum];

	// SQL命令
	_SqlCommand := 
//	'INSERT INTO msg (msgtime, msg_level, msgnum, str1, str2) VALUES ({msgtime}, {msg_level}, {msgnum}, {str1})';

	'INSERT INTO msg (su, msgtime, msg_level, msgnum, str1, str2, raw_msg_str) VALUES (uuidV7(), {msgtime}::timestamptz, {msg_level}, {msgnum}, {str1}, {str2}, {raw_msg_str})';

	msgtmp.msgTIME := msg.msgTIME;
	msgtmp.Level := msg.Level;
	msgtmp.Number := msg.Number;

	str := ADR(msg.MsgStr1);
	msgtmp.MsgStr1 := str^;

	str2 := ADR(msg.MsgStr2);
	msgtmp.MsgStr2 := str2^;

	str3 := ADR(msg.raw_msg_str);
	msgtmp.raw_msg_str := str3^;


// 設定對應參數
	_stPara[0].sParaName := 'msgtime'; 		_stPara[0].eParaType := E_ExpParameterType.DateTime; 	_stPara[0].nParaSize := SIZEOF(msgtmp.msgTIME);
	_stPara[1].sParaName := 'msg_level'; 	_stPara[1].eParaType := E_ExpParameterType.Int16; 		_stPara[1].nParaSize := SIZEOF(msgtmp.Level);
	_stPara[2].sParaName := 'msgnum';		_stPara[2].eParaType := E_ExpParameterType.Int16;		_stPara[2].nParaSize := SIZEOF(msgtmp.Number);
	_stPara[3].sParaName := 'str1';			_stPara[3].eParaType := E_ExpParameterType.WSTRING_;	_stPara[3].nParaSize := 160;
	_stPara[4].sParaName := 'str2';			_stPara[4].eParaType := E_ExpParameterType.WSTRING_;	_stPara[4].nParaSize := 160;
	_stPara[5].sParaName := 'raw_msg_str';	_stPara[5].eParaType := E_ExpParameterType.WSTRING_;	_stPara[5].nParaSize := 500;


	IF 
		_fb_PLCDBCmdEvt.Execute(
			hDBID := 1,
			pExpression := ADR(_SqlCommand),			// SQL 命令 ex. SELECT * FROM PlcTest.newtable WHERE ID = {ID}  
			cbExpression := SIZEOF(_SqlCommand),		// SQL 命令字串的長度
			pData:= ADR(msgtmp),		// 帶入的參數值
			cbData:= SIZEOF(msgtmp),//itmp, 	// 帶入的參數值大小
			pParameter:= ADR(_stPara), 				// 帶入的參數類型設定  ex.上面命令內的 {ID} 類型設定
			cbParameter:= SIZEOF(_stPara),			// 帶入的參數類型設定的大小
		) 
	THEN
		IF _fb_PLCDBCmdEvt.bError THEN
			tcMessage := _fb_PLCDBCmdEvt.ipTcResult;
		END_IF
		msgbuff.DoneNumber := msgbuff.DoneNumber + 1;
	END_IF
ELSIF msgbuff.DoneNumber > msgbuff.evenNumber THEN
	msgbuff.DoneNumber := msgbuff.evenNumber;
END_IF

MsgBuff.systime(
	bEnable:= TRUE, 
	dwCycle:= 1,
	systemTime=> );
MsgBuff.currentTime := SYSTEMTIME_TO_DT(MsgBuff.systime.systemTime);

END_PROGRAM

// ---- POUs/功能塊/字串處理功能塊/字串連接/WStrConcat.TcPOU
FUNCTION WStrConcat : WSTRING(511)
VAR_INPUT
	str0 : WSTRING(511) := "";
	str1 : WSTRING(511) := "";
	str2 : WSTRING(511) := "";
	str3 : WSTRING(511) := "";
	str4 : WSTRING(511) := "";
	str5 : WSTRING(511) := "";
	str6 : WSTRING(511) := "";
	str7 : WSTRING(511) := "";
	str8 : WSTRING(511) := "";
END_VAR
VAR
	tmpstr : WSTRING(511);
END_VAR

tmpstr := WCONCAT(STR1:= str0, STR2:= str1);
tmpstr := WCONCAT(STR1:= tmpstr, STR2:= str2);
tmpstr := WCONCAT(STR1:= tmpstr, STR2:= str3);
tmpstr := WCONCAT(STR1:= tmpstr, STR2:= str4);
tmpstr := WCONCAT(STR1:= tmpstr, STR2:= str5);
tmpstr := WCONCAT(STR1:= tmpstr, STR2:= str6);
tmpstr := WCONCAT(STR1:= tmpstr, STR2:= str7);
tmpstr := WCONCAT(STR1:= tmpstr, STR2:= str8);
WStrConcat := tmpstr;
RETURN;

END_FUNCTION

// ---- POUs/硬體控制/油壓系統/Hydraulic.TcPOU
PROGRAM Hydraulic
VAR
	// 臺車升降用
	step : INT;
	// 靠邊用
	step1 : INT;
	
	ActionMode : Hydraulic_Action;
	
	// 升降動作的台車 bit0:台車1 bit1:台車2 bit2:台車3 bit3:台車4
	CarLift_Select : WORD;
	
	// 升降動作等待繼續 bit0:台車1 bit1:台車2 bit2:台車3 bit3:台車4
	CarLift_WaitSync : WORD;
	
	tmr01: TON;
	
	tmr1_01: TON;
	tmr1_02: TON;
	
	StepA : INT;
	StepB : INT;
	StepC : INT;
	StepD : INT;
	
	tmrA_1: TON;
	tmrA_10: TON;
	tmrB_1: TON;
	tmrB_10: TON;
	tmrC_1: TON;
	tmrC_10: TON;
	tmrD_1: TON;
	tmrD_10: TON;
	
	tmr_pump: TON;
	
	TryCount: INT;
END_VAR


VAR_OUTPUT
	bDone: BOOL;
	bBuzy: BOOL;
	bError: BOOL;
	
	bDone1: BOOL;
	bBuzy1: BOOL;
	bError1: BOOL;
END_VAR

IF (EStop OR SystemError) AND bBuzy THEN
	IF bBuzy THEN
		step := step  + 10000;
	END_IF
	io.q101 := FALSE;
	io.q301 := FALSE;
	io.q201 := FALSE;
	io.q202 := FALSE;
	io.q203 := FALSE;
	io.q204 := FALSE;
	io.q205 := FALSE;
	io.q206 := FALSE;
	io.q207 := FALSE;
	io.q208 := FALSE;
	io.q302 := FALSE;
END_IF


// 
Step_0_Start();
Step_1_Stop();
step_2_CarLift_Up();
step_4_CarLift_Mid();
step_6_CarLift_Down();

step1_1_Pull_over();
step1_2_Pull_over_Jog();

bBuzy := step > 0 AND step < 10000;
bError := step > 10000;

IF bError OR bBuzy THEN
	bDone := FALSE;
END_IF

bBuzy1 := step1 > 0 AND step1 < 10000;
bError1 := step1 > 10000;

IF bError1 OR bBuzy1 THEN
	bDone1 := FALSE;
END_IF


// 油壓未使用關閉計時器
tmr_pump.in := NOT(bBuzy OR bBuzy1) AND io.q101;
tmr_pump.pt := T#1M;

IF tmr_pump.q THEN
	io.q101 := FALSE;
	io.q301 := FALSE;
END_IF

tmrAct();

METHOD CarLift_Down : BOOL
VAR_INPUT
	// 動作的台車 bit0:台車1、bit0:台車2、bit0:台車3、bit0:台車4
	Action_Select : WORD := 0;
END_VAR
ActionMode := Hydraulic_Action.Car_2_Dn;

CarLift_Select := Action_Select;

step := 1;
END_METHOD

METHOD CarLift_Mid : BOOL
VAR_INPUT
	// 動作的台車 bit0:台車1、bit0:台車2、bit0:台車3、bit0:台車4
	Action_Select : WORD := 0;
END_VAR
ActionMode := Hydraulic_Action.Car_2_Mid;

CarLift_Select := Action_Select;

step := 1;
END_METHOD

METHOD CarLift_Up : BOOL
VAR_INPUT
	// 動作的台車 bit0:台車1、bit0:台車2、bit0:台車3、bit0:台車4
	Action_Select : WORD := 0;
END_VAR
ActionMode := Hydraulic_Action.Car_2_Up;

CarLift_Select := Action_Select;

step := 1;
END_METHOD

ACTION io_ref:

END_ACTION

// 靠邊油壓動作
METHOD Over_Pull : BOOL
VAR_INPUT
	// 使用的感應器 感應器1 : 2,300mm  感應器2 : X 感應器2 : 6,080mm  感應器3 : 10,230mm 
	Leageth : INT;
END_VAR
VAR
	Select_tmp:WORD;
END_VAR
ActionMode := Hydraulic_Action.Pull_over;

Select_tmp := 0;

Select_tmp.0 := Leageth > 2300;
Select_tmp.1 := FALSE;
Select_tmp.2 := Leageth > 6080;
Select_tmp.3 := Leageth > 10230;

CarLift_Select := Select_tmp;

IF NOT io.q101 THEN
	step := 1;
ELSE
	step1 := 100;
END_IF
END_METHOD

// 靠邊油壓動作
METHOD Over_Pull_Jog : BOOL
VAR_INPUT
END_VAR
ActionMode := Hydraulic_Action.Pull_over_Jog;

IF NOT io.q101 THEN
	step := 1;
ELSE
	step1 := 200;
END_IF
END_METHOD

ACTION Step_0_Start:
CASE step OF
	1:// 檢查油壓泵狀態
		IF io.i102 THEN
			// !!錯誤!! 油壓泵馬達過載
			step := step + 10000;
		ELSIF io.i104 THEN
			// !!錯誤!! 油壓泵馬達過載
			step := step + 10000;
		ELSE
			step := step + 1;
		END_IF
		
	2:
		
		step := 10;
		
	10: // 如果油壓流已經啟動，則跳過
		IF io.q101 THEN
			step := 20;
		ELSE
			step := step + 1;
		END_IF
		
	11:// 啟動油壓泵
		io.q101 := TRUE;
		step := step + 1;
		
	12:
		tmr01.PT := T#1S;
		tmr01.in := TRUE;
		IF tmr01.q THEN
			tmr01.in := FALSE;
			step := step + 1;
		END_IF
		
	13:
		step := 20;
		
	20:
		step := 80;
		
	80:
		CASE ActionMode OF
			Hydraulic_Action.Car_2_Up:
				Step := 200;
			
			Hydraulic_Action.Car_2_Mid:
				step := 400;
				
			Hydraulic_Action.Car_2_dn:
				step := 600;
				
			Hydraulic_Action.Pull_over:
				io.q301 := TRUE;
				step1 := 100;
				step := 0;
				
			Hydraulic_Action.Pull_over_Jog:
				io.q301 := TRUE;
				step1 := 200;
				step := 0;
				
		END_CASE
END_CASE
END_ACTION

ACTION Step_1_Stop:
CASE step OF
	100:
		io.q201 := FALSE;
		io.q202 := FALSE;
		io.q203 := FALSE;
		io.q204 := FALSE;
		io.q205 := FALSE;
		io.q206 := FALSE;
		io.q207 := FALSE;
		io.q208 := FALSE;
		
		stepA := 0;
		stepB := 0;
		stepC := 0;
		stepD := 0;
		
		io.q301 := FALSE;
		io.q302 := FALSE;
		
		tmr01.IN :=FALSE;
		step := step + 1;
		
	101:
		step := 0;
		
END_CASE
END_ACTION

ACTION step_2_CarLift_Up:
CASE step OF
	200:
		
		IF (CarLift_Select AND 16#F) = 0 THEN
			CarLift_Select := 15;
		END_IF
		step := step + 1;
	
	201:
		io.q301 := TRUE;
		IF CarLift_Select.0 THEN
			stepA := 200;
		END_IF
		
		IF CarLift_Select.1 THEN
			stepB := 200;
		END_IF
		
		IF CarLift_Select.2 THEN
			stepC := 200;
		END_IF
		
		IF CarLift_Select.3 THEN
			stepD := 200;
		END_IF
		
		step := step + 1;
		
	202:
		IF stepA = 0 AND stepB = 0 AND stepC = 0 AND stepD = 0 THEN
			step := step + 1;
		ELSIF stepA > 10000 OR stepB > 10000 OR stepC > 10000 OR stepD > 10000 THEN
			step := step + 10000;
		END_IF
		
	203:
		io.q301 := false;
		CarLift_Select := 0;
		bDone := TRUE;
		step := 0;
		
END_CASE

{region "============= 台車A上升  ============="}
CASE stepA OF
	200: // 啟動上升
		io.q201 := TRUE;
		io.q202 := FALSE;
		stepA := stepA + 1;
		
	201: // 啟動超時計時器
		tmrA_10.PT := T#20S;
		tmrA_10.IN := TRUE;
		stepA := stepA + 1;
		
	202: // 等待
		IF NOT io.i201 OR tmrA_10.q THEN
			tmrA_10.in := FALSE;
			IF NOT io.i201 THEN
				stepA := stepA + 1;
			ELSIF tmrA_10.q THEN
				io.q201 := FALSE;
				stepA := stepA + 10000;
			END_IF
		END_IF
		
	203: // 成功之後等待1秒
		tmrA_1.PT := T#1S;
		tmrA_1.IN := TRUE;
		IF tmrA_1.Q THEN
		 	io.q201 := FALSE;
			stepA := stepA + 1;
		END_IF
		
	204:
		stepA := 0;
		
END_CASE
{endregion}

{region "============= 台車B上升  ============="}
CASE stepB OF
	200: // 啟動上升
		io.q203 := TRUE;
		io.q204 := FALSE;
		stepB := stepB + 1;
		
	201: // 啟動超時計時器
		tmrB_10.PT := T#20S;
		tmrB_10.IN := TRUE;
		stepB := stepB + 1;
		
	202: // 等待
		IF NOT io.i204 OR tmrB_10.q THEN
			
			tmrB_10.in := FALSE;
			
			IF NOT io.i204 THEN
				stepB := stepB + 1;
			ELSIF tmrB_10.q THEN
				io.q203 := FALSE;
				stepB := stepB + 10000;
			END_IF
		END_IF
		
	203: // 成功之後等待1秒
		tmrB_1.PT := T#1S;
		tmrB_1.IN := TRUE;
		IF tmrB_1.Q THEN
			io.q203 := FALSE;
			stepB := stepB + 1;
		END_IF
		
	204:
		stepB := 0;
		
END_CASE
{endregion}

{region "============= 台車C上升  ============="}
CASE stepC OF
	200: // 啟動上升
		io.q205 := TRUE;
		io.q206 := FALSE;
		stepC := stepC + 1;
		
	201: // 啟動超時計時器
		tmrC_10.PT := T#20S;
		tmrC_10.IN := TRUE;
		stepC := stepC + 1;
		
	202: // 等待
		IF NOT io.i207 OR tmrC_10.q THEN
			tmrC_10.in := FALSE;
			
			IF NOT io.i207 THEN
				stepC := stepC + 1;
			ELSIF tmrC_10.q THEN
				io.q205 := FALSE;
				stepC := stepC + 10000;
			END_IF
		END_IF
		
	203: // 成功之後等待1秒
		tmrC_1.PT := T#1S;
		tmrC_1.IN := TRUE;
		IF tmrC_1.Q THEN
			io.q205 := FALSE;
			stepC := stepC + 1;
		END_IF
		
	204:
		stepC := 0;
		
END_CASE
{endregion}

{region "============= 台車D上升  ============="}
CASE stepD OF
	200: // 啟動上升
		io.q207 := TRUE;
		io.q208 := FALSE;
		stepD := stepD + 1;
		
	201: // 啟動超時計時器
		tmrD_10.PT := T#20S;
		tmrD_10.IN := TRUE;
		stepD := stepD + 1;
		
	202: // 等待
		IF NOT io.i210 OR tmrD_10.q THEN
			tmrD_10.in := FALSE;
			
			IF NOT io.i210 THEN
				stepD := stepD + 1;
			ELSIF tmrD_10.q THEN
				io.q207 := FALSE;
				stepD := stepD + 10000;
			END_IF
		END_IF
		
	203: // 成功之後等待1秒
		tmrD_1.PT := T#1S;
		tmrD_1.IN := TRUE;
		IF tmrD_1.Q THEN
			io.q207 := FALSE;
			stepD := stepD + 1;
		END_IF
		
	204:
		stepD := 0;
		
END_CASE
{endregion}
END_ACTION

ACTION step_4_CarLift_Mid:
CASE step OF
	400:
		CarLift_WaitSync := 0;
		IF (CarLift_Select AND 16#F) = 0 THEN
			CarLift_Select := 15;
		END_IF
		step := step + 1;
	
	401:
		io.q301 := TRUE;
		IF CarLift_Select.0 THEN
			stepA := 400;
		END_IF
		
		IF CarLift_Select.1 THEN
			stepB := 400;
		END_IF
		
		IF CarLift_Select.2 THEN
			stepC := 400;
		END_IF
		
		IF CarLift_Select.3 THEN
			stepD := 400;
		END_IF
		
		step := step + 1;
		
	402:
		IF stepA = 0 AND stepB = 0 AND stepC = 0 AND stepD = 0 THEN
			step := 420;
		ELSIF CarLift_WaitSync = CarLift_Select THEN
			step := 410;
		ELSIF stepA > 10000 OR stepB > 10000 OR stepC > 10000 OR stepD > 10000 THEN
			step := step + 10000;
		END_IF
		
	410: // 切換成慢速模式
		io.q301 := FALSE;
		step := step + 1;
		
	411:
		tmr01.PT := T#1S;
		tmr01.in := TRUE;
		IF tmr01.q THEN
			tmr01.in := FALSE;
			step := step + 1;
		END_IF
		
	412:IF CarLift_Select.0 THEN
			stepA := stepA + 1;
		END_IF
		
		IF CarLift_Select.1 THEN
			stepB := stepB + 1;
		END_IF
		
		IF CarLift_Select.2 THEN
			stepC := stepC + 1;
		END_IF
		
		IF CarLift_Select.3 THEN
			stepD := stepD + 1;
		END_IF
		step := step + 1;
		
	413:
		step := 420;
		
	420:
		io.q301 := FALSE;
		CarLift_Select := 0;
		bDone := TRUE;
		step := 0;
		
END_CASE

{region "============= 台車A中位移動  ============="}
CASE stepA OF
	400: // 判斷位置
		IF NOT io.i202 THEN
			stepA := 0;
		ELSE
			IF NOT io.i201 THEN
				// 位置在上限
				stepA := 410;
			ELSIF NOT io.i203 THEN
				// 位置在下限
				stepA := 440;
			ELSE
			    // 位置不確定
				stepA := 470;
		 	END_IF
		END_IF
	{region "============= 位置在上限  ============="}	
	410: // 位置在上限，下降
		io.q201 := FALSE;
		io.q202 := TRUE;
		stepA := stepA + 1;
			 
	411:
		tmrA_10.PT := T#60S;
		tmrA_10.IN := TRUE;
		stepA := stepA + 1;
			 
	412://
		IF NOT io.i202 OR tmrA_10.q THEN
			tmrA_10.in := FALSE;
			IF NOT io.i202 THEN
				stepA := stepA + 1;
			ELSIF tmrA_10.q THEN
				stepA := stepA + 10000;
			END_IF
		END_IF
			 
	413: // 先降過頭在慢速升回
		IF io.i202 THEN
			io.q202 := FALSE;
			stepA := stepA + 1;
		END_IF
				  
	414:
		CarLift_WaitSync.0 := TRUE;
		stepA := 420;
				  
//	420: // 等待主油壓切至慢速模式 ，完成後由主流程跳步
		
				  
	421: // 用慢速上升
		io.q201 := TRUE;
		IF NOT io.i202 THEN
			io.q201 := FALSE;
			stepA := stepA + 1;
		END_IF
				  
	422: // 用慢速上升
		io.q201 := TRUE;
		IF NOT io.i202 THEN
			io.q201 := FALSE;
			stepA := stepA + 1;
		END_IF
		
	423:
		stepA := 0;
	{endregion}
	{region "============= 位置在下限  ============="}	
	440: // 位置在下限，上升
		io.q201 := TRUE;
		io.q202 := FALSE;
		stepA := stepA + 1;
			 
